LIN {X 0,Y 358.21,Z 356.559,A -85,B 0,C 180,E1 -13447.914,E2 -13447.914} C_VEL
LIN {X 0,Y 359.231,Z 351.066,A -85,B 0,C 180,E1 -13450.213,E2 -13450.213} C_VEL
LIN {X 0,Y 358.495,Z 346.197,A -85,B 0,C 180,E1 -13452.681,E2 -13452.681} C_VEL
LIN {X 0,Y 357.44,Z 341.043,A -85,B 0,C 180,E1 -13455.752,E2 -13455.752} C_VEL
LIN {X 0,Y 356.358,Z 336.09,A -85,B 0,C 180,E1 -13459.397,E2 -13459.397} C_VEL
LIN {X 0,Y 355.734,Z 333.05,A -85,B 0,C 180,E1 -13462.234,E2 -13462.234} C_VEL
LIN {X 0,Y 355.208,Z 330.772,A -85,B 0,C 180,E1 -13464.986,E2 -13464.986} C_VEL
LIN {X 0,Y 354.793,Z 328.931,A -85,B 0,C 180,E1 -13468.088,E2 -13468.088} C_VEL
LIN {X 0,Y 354.858,Z 329.119,A -85,B 0,C 180,E1 -13470.427,E2 -13470.427} C_VEL
LIN {X 0,Y 355.199,Z 330.372,A -85,B 0,C 180,E1 -13470.749,E2 -13470.749} C_VEL
LIN {X 0,Y 356.216,Z 332.283,A -85,B 0,C 180,E1 -13471.122,E2 -13471.122} C_VEL
LIN {X 0,Y 357.49,Z 333.609,A -85,B 0,C 180,E1 -13471.474,E2 -13471.474} C_VEL
LIN {X 0,Y 358.898,Z 336.455,A -85,B 0,C 180,E1 -13471.968,E2 -13471.968} C_VEL
LIN {X 0,Y 362.469,Z 342.56,A -85,B 0,C 180,E1 -13473.115,E2 -13473.115} C_VEL
LIN {X 0,Y 366.125,Z 350.503,A -85,B 0,C 180,E1 -13474.449,E2 -13474.449} C_VEL
LIN {X 0,Y 369.455,Z 359.944,A -85,B 0,C 180,E1 -13475.937,E2 -13475.937} C_VEL
LIN {X 0,Y 370.427,Z 363.82,A -85,B 0,C 180,E1 -13476.52,E2 -13476.52} C_VEL
LIN {X 0,Y 368.443,Z 376.173,A -85,B 0,C 180,E1 -13477.869,E2 -13477.869} C_VEL
LIN {X 0,Y 366.706,Z 386.37,A -85,B 0,C 180,E1 -13479.234,E2 -13479.234} C_VEL
LIN {X 0,Y 364.738,Z 396.604,A -85,B 0,C 180,E1 -13480.879,E2 -13480.879} C_VEL
LIN {X 0,Y 362.547,Z 406.465,A -85,B 0,C 180,E1 -13482.805,E2 -13482.805} C_VEL
LIN {X 0,Y 360.903,Z 414.416,A -85,B 0,C 180,E1 -13484.759,E2 -13484.759} C_VEL
LIN {X 0,Y 359.55,Z 419.998,A -85,B 0,C 180,E1 -13486.435,E2 -13486.435} C_VEL
LIN {X 0,Y 358.205,Z 425.911,A -85,B 0,C 180,E1 -13488.685,E2 -13488.685} C_VEL
LIN {X 0,Y 356.995,Z 430.235,A -85,B 0,C 180,E1 -13490.939,E2 -13490.939} C_VEL
LIN {X 0,Y 356.046,Z 433.125,A -85,B 0,C 180,E1 -13493.199,E2 -13493.199} C_VEL
LIN {X 0,Y 355.518,Z 434.622,A -85,B 0,C 180,E1 -13495.465,E2 -13495.465} C_VEL
LIN {X 0,Y 355.148,Z 434.801,A -85,B 0,C 180,E1 -13497.732,E2 -13497.732} C_VEL
LIN {X 0,Y 354.952,Z 433.645,A -85,B 0,C 180,E1 -13500,E2 -13500} C_VEL
LIN {X 0,Y 354.878,Z 431.132,A -85,B 0,C 180,E1 -13502.27,E2 -13502.27} C_VEL
LIN {X 0,Y 354.897,Z 427.195,A -85,B 0,C 180,E1 -13504.544,E2 -13504.544} C_VEL
LIN {X 0,Y 355.363,Z 423.255,A -85,B 0,C 180,E1 -13506.245,E2 -13506.245} C_VEL
LIN {X 0,Y 355.737,Z 418.361,A -85,B 0,C 180,E1 -13507.949,E2 -13507.949} C_VEL
LIN {X 0,Y 356.3,Z 411.398,A -85,B 0,C 180,E1 -13509.939,E2 -13509.939} C_VEL
LIN {X 0,Y 357.101,Z 402.834,A -85,B 0,C 180,E1 -13511.926,E2 -13511.926} C_VEL
LIN {X 0,Y 357.899,Z 393.943,A -85,B 0,C 180,E1 -13513.63,E2 -13513.63} C_VEL
LIN {X 0,Y 358.893,Z 383.272,A -85,B 0,C 180,E1 -13515.329,E2 -13515.329} C_VEL
LIN {X 0,Y 359.931,Z 372.22,A -85,B 0,C 180,E1 -13516.794,E2 -13516.794} C_VEL
LIN {X 0,Y 360.928,Z 359.901,A -85,B 0,C 180,E1 -13518.153,E2 -13518.153} C_VEL
LIN {X 0,Y 361.541,Z 352.454,A -85,B 0,C 180,E1 -13518.855,E2 -13518.855} C_VEL
LIN {X 0,Y 358.245,Z 340.353,A -85,B 0,C 180,E1 -13520.025,E2 -13520.025} C_VEL
LIN {X 0,Y 354.959,Z 329.484,A -85,B 0,C 180,E1 -13520.98,E2 -13520.98} C_VEL
LIN {X 0,Y 354.871,Z 328.937,A -85,B 0,C 180,E1 -13521.207,E2 -13521.207} C_VEL
LIN {X 0,Y 354.867,Z 328.909,A -85,B 0,C 180,E1 -13524.576,E2 -13524.576} C_VEL
LIN {X 0,Y 354.889,Z 328.902,A -85,B 0,C 180,E1 -13527.096,E2 -13527.096} C_VEL
LIN {X 0,Y 354.859,Z 328.904,A -85,B 0,C 180,E1 -13529.679,E2 -13529.679} C_VEL
LIN {X 0,Y 354.811,Z 328.91,A -85,B 0,C 180,E1 -13533.702,E2 -13533.702} C_VEL
LIN {X 0,Y 354.803,Z 328.916,A -85,B 0,C 180,E1 -13536.459,E2 -13536.459} C_VEL
LIN {X 0,Y 354.829,Z 328.907,A -85,B 0,C 180,E1 -13539.424,E2 -13539.424} C_VEL
LIN {X 0,Y 354.793,Z 328.914,A -85,B 0,C 180,E1 -13542.867,E2 -13542.867} C_VEL
LIN {X 0,Y 354.782,Z 328.916,A -85,B 0,C 180,E1 -13546.105,E2 -13546.105} C_VEL
LIN {X 0,Y 354.83,Z 328.908,A -85,B 0,C 180,E1 -13549.184,E2 -13549.184} C_VEL
LIN {X 0,Y 354.818,Z 328.914,A -85,B 0,C 180,E1 -13552.401,E2 -13552.401} C_VEL
LIN {X 0,Y 354.818,Z 328.91,A -85,B 0,C 180,E1 -13554.941,E2 -13554.941} C_VEL
LIN {X 0,Y 354.799,Z 328.916,A -85,B 0,C 180,E1 -13558.405,E2 -13558.405} C_VEL
LIN {X 0,Y 354.852,Z 328.906,A -85,B 0,C 180,E1 -13561.618,E2 -13561.618} C_VEL
LIN {X 0,Y 354.904,Z 328.904,A -85,B 0,C 180,E1 -13564.172,E2 -13564.172} C_VEL
LIN {X 0,Y 354.821,Z 328.913,A -85,B 0,C 180,E1 -13567.892,E2 -13567.892} C_VEL
LIN {X 0,Y 354.929,Z 328.9,A -85,B 0,C 180,E1 -13571.891,E2 -13571.891} C_VEL
LIN {X 0,Y 354.949,Z 328.899,A -85,B 0,C 180,E1 -13575.98,E2 -13575.98} C_VEL
LIN {X 0,Y 354.983,Z 328.893,A -85,B 0,C 180,E1 -13579.735,E2 -13579.735} C_VEL
LIN {X 0,Y 355.119,Z 328.876,A -85,B 0,C 180,E1 -13582.036,E2 -13582.036} C_VEL
LIN {X 0,Y 355.096,Z 328.876,A -85,B 0,C 180,E1 -13584.32,E2 -13584.32} C_VEL
LIN {X 0,Y 355.249,Z 328.861,A -85,B 0,C 180,E1 -13587.731,E2 -13587.731} C_VEL
LIN {X 0,Y 355.401,Z 328.84,A -85,B 0,C 180,E1 -13589.999,E2 -13589.999} C_VEL
LIN {X 0,Y 355.248,Z 328.856,A -85,B 0,C 180,E1 -13592.267,E2 -13592.267} C_VEL
LIN {X 0,Y 355.143,Z 328.869,A -85,B 0,C 180,E1 -13596.818,E2 -13596.818} C_VEL
LIN {X 0,Y 355.019,Z 328.885,A -85,B 0,C 180,E1 -13599.111,E2 -13599.111} C_VEL
LIN {X 0,Y 354.924,Z 328.896,A -85,B 0,C 180,E1 -13602.58,E2 -13602.58} C_VEL
LIN {X 0,Y 354.892,Z 328.901,A -85,B 0,C 180,E1 -13606.095,E2 -13606.095} C_VEL
LIN {X 0,Y 354.903,Z 328.898,A -85,B 0,C 180,E1 -13608.471,E2 -13608.471} C_VEL
LIN {X 0,Y 354.837,Z 328.907,A -85,B 0,C 180,E1 -13612.105,E2 -13612.105} C_VEL
LIN {X 0,Y 354.9,Z 328.9,A -85,B 0,C 180,E1 -13615.826,E2 -13615.826} C_VEL
LIN {X 0,Y 354.817,Z 328.911,A -85,B 0,C 180,E1 -13619.68,E2 -13619.68} C_VEL
LIN {X 0,Y 354.805,Z 328.912,A -85,B 0,C 180,E1 -13623.701,E2 -13623.701} C_VEL
LIN {X 0,Y 354.796,Z 328.912,A -85,B 0,C 180,E1 -13626.458,E2 -13626.458} C_VEL
LIN {X 0,Y 354.822,Z 328.912,A -85,B 0,C 180,E1 -13629.422,E2 -13629.422} C_VEL
LIN {X 0,Y 354.786,Z 328.917,A -85,B 0,C 180,E1 -13632.866,E2 -13632.866} C_VEL
LIN {X 0,Y 354.773,Z 328.914,A -85,B 0,C 180,E1 -13636.104,E2 -13636.104} C_VEL
LIN {X 0,Y 354.774,Z 328.916,A -85,B 0,C 180,E1 -13639.533,E2 -13639.533} C_VEL
LIN {X 0,Y 354.116,Z 329,A -85,B 0,C 180,E1 -13640.481,E2 -13640.481} C_VEL
LIN {X 0,Y 351.3,Z 329.347,A -85,B 0,C 180,E1 -13642.024,E2 -13642.024} C_VEL
LIN {X 0,Y 348.899,Z 329.649,A -85,B 0,C 180,E1 -13643.272,E2 -13643.272} C_VEL
LIN {X 0,Y 347.846,Z 329.778,A -85,B 0,C 180,E1 -13644.237,E2 -13644.237} C_VEL
LIN {X 0,Y 347.748,Z 329.787,A -85,B 0,C 180,E1 -13644.564,E2 -13644.564} C_VEL
LIN {X 0,Y 347.759,Z 329.789,A -85,B 0,C 180,E1 -13648.301,E2 -13648.301} C_VEL
LIN {X 0,Y 347.801,Z 329.787,A -85,B 0,C 180,E1 -13650.989,E2 -13650.989} C_VEL
LIN {X 0,Y 347.826,Z 329.78,A -85,B 0,C 180,E1 -13653.607,E2 -13653.607} C_VEL
LIN {X 0,Y 347.783,Z 329.786,A -85,B 0,C 180,E1 -13656.161,E2 -13656.161} C_VEL
LIN {X 0,Y 347.806,Z 329.783,A -85,B 0,C 180,E1 -13659.909,E2 -13659.909} C_VEL
LIN {X 0,Y 347.859,Z 329.779,A -85,B 0,C 180,E1 -13662.358,E2 -13662.358} C_VEL
LIN {X 0,Y 347.89,Z 329.773,A -85,B 0,C 180,E1 -13665.97,E2 -13665.97} C_VEL
LIN {X 0,Y 347.921,Z 329.768,A -85,B 0,C 180,E1 -13669.525,E2 -13669.525} C_VEL
LIN {X 0,Y 348.1,Z 329.747,A -85,B 0,C 180,E1 -13673.042,E2 -13673.042} C_VEL
LIN {X 0,Y 348.201,Z 329.734,A -85,B 0,C 180,E1 -13677.686,E2 -13677.686} C_VEL
LIN {X 0,Y 348.338,Z 329.718,A -85,B 0,C 180,E1 -13680,E2 -13680} C_VEL
LIN {X 0,Y 348.201,Z 329.739,A -85,B 0,C 180,E1 -13682.313,E2 -13682.313} C_VEL
LIN {X 0,Y 348.098,Z 329.747,A -85,B 0,C 180,E1 -13686.958,E2 -13686.958} C_VEL
LIN {X 0,Y 347.961,Z 329.763,A -85,B 0,C 180,E1 -13689.298,E2 -13689.298} C_VEL
LIN {X 0,Y 347.886,Z 329.773,A -85,B 0,C 180,E1 -13692.839,E2 -13692.839} C_VEL
LIN {X 0,Y 347.833,Z 329.782,A -85,B 0,C 180,E1 -13696.431,E2 -13696.431} C_VEL
LIN {X 0,Y 347.848,Z 329.777,A -85,B 0,C 180,E1 -13698.86,E2 -13698.86} C_VEL
LIN {X 0,Y 347.766,Z 329.789,A -85,B 0,C 180,E1 -13702.58,E2 -13702.58} C_VEL
LIN {X 0,Y 347.804,Z 329.783,A -85,B 0,C 180,E1 -13705.109,E2 -13705.109} C_VEL
LIN {X 0,Y 347.805,Z 329.786,A -85,B 0,C 180,E1 -13707.694,E2 -13707.694} C_VEL
LIN {X 0,Y 347.763,Z 329.79,A -85,B 0,C 180,E1 -13710.346,E2 -13710.346} C_VEL
LIN {X 0,Y 347.741,Z 329.795,A -85,B 0,C 180,E1 -13714.044,E2 -13714.044} C_VEL
LIN {X 0,Y 347.76,Z 329.793,A -85,B 0,C 180,E1 -13717.321,E2 -13717.321} C_VEL
LIN {X 0,Y 347.86,Z 330.034,A -85,B 0,C 180,E1 -13719.537,E2 -13719.537} C_VEL
LIN {X 0,Y 349.468,Z 338.436,A -85,B 0,C 180,E1 -13723.138,E2 -13723.138} C_VEL
LIN {X 0,Y 351.233,Z 347.023,A -85,B 0,C 180,E1 -13726.645,E2 -13726.645} C_VEL
LIN {X 0,Y 352.492,Z 353.68,A -85,B 0,C 180,E1 -13729.257,E2 -13729.257} C_VEL
LIN {X 0,Y 352.257,Z 357.86,A -85,B 0,C 180,E1 -13730.782,E2 -13730.782} C_VEL
LIN {X 0,Y 350.874,Z 368.306,A -85,B 0,C 180,E1 -13734.49,E2 -13734.49} C_VEL
LIN {X 0,Y 349.619,Z 379.808,A -85,B 0,C 180,E1 -13738.491,E2 -13738.491} C_VEL
LIN {X 0,Y 348.526,Z 391.621,A -85,B 0,C 180,E1 -13742.53,E2 -13742.53} C_VEL
LIN {X 0,Y 347.843,Z 402.269,A -85,B 0,C 180,E1 -13746.072,E2 -13746.072} C_VEL
LIN {X 0,Y 348.261,Z 406.952,A -85,B 0,C 180,E1 -13746.317,E2 -13746.317} C_VEL
LIN {X 0,Y 350.008,Z 423.225,A -85,B 0,C 180,E1 -13747.11,E2 -13747.11} C_VEL
LIN {X 0,Y 351.474,Z 437.917,A -85,B 0,C 180,E1 -13748.059,E2 -13748.059} C_VEL
LIN {X 0,Y 352.452,Z 450.642,A -85,B 0,C 180,E1 -13749.077,E2 -13749.077} C_VEL
LIN {X 0,Y 352.517,Z 455.971,A -85,B 0,C 180,E1 -13749.557,E2 -13749.557} C_VEL
LIN {X 0,Y 351.156,Z 468.911,A -85,B 0,C 180,E1 -13750.87,E2 -13750.87} C_VEL
LIN {X 0,Y 349.938,Z 480.529,A -85,B 0,C 180,E1 -13752.317,E2 -13752.317} C_VEL
LIN {X 0,Y 348.836,Z 491.162,A -85,B 0,C 180,E1 -13753.919,E2 -13753.919} C_VEL
LIN {X 0,Y 347.921,Z 500.982,A -85,B 0,C 180,E1 -13755.705,E2 -13755.705} C_VEL
LIN {X 0,Y 347.322,Z 510.138,A -85,B 0,C 180,E1 -13757.734,E2 -13757.734} C_VEL
LIN {X 0,Y 347.071,Z 516.625,A -85,B 0,C 180,E1 -13759.501,E2 -13759.501} C_VEL
LIN {X 0,Y 347.029,Z 521.956,A -85,B 0,C 180,E1 -13761.265,E2 -13761.265} C_VEL
LIN {X 0,Y 347.145,Z 526.251,A -85,B 0,C 180,E1 -13763.024,E2 -13763.024} C_VEL
LIN {X 0,Y 347.243,Z 528.547,A -85,B 0,C 180,E1 -13764.193,E2 -13764.193} C_VEL
LIN {X 0,Y 347.327,Z 530.421,A -85,B 0,C 180,E1 -13765.359,E2 -13765.359} C_VEL
LIN {X 0,Y 347.494,Z 532.968,A -85,B 0,C 180,E1 -13767.683,E2 -13767.683} C_VEL
LIN {X 0,Y 347.652,Z 533.671,A -85,B 0,C 180,E1 -13768.843,E2 -13768.843} C_VEL
LIN {X 0,Y 347.813,Z 533.994,A -85,B 0,C 180,E1 -13770.001,E2 -13770.001} C_VEL
LIN {X 0,Y 347.636,Z 533.883,A -85,B 0,C 180,E1 -13771.159,E2 -13771.159} C_VEL
LIN {X 0,Y 347.32,Z 532.528,A -85,B 0,C 180,E1 -13773.481,E2 -13773.481} C_VEL
LIN {X 0,Y 347.26,Z 531.296,A -85,B 0,C 180,E1 -13774.644,E2 -13774.644} C_VEL
LIN {X 0,Y 346.944,Z 527.65,A -85,B 0,C 180,E1 -13776.982,E2 -13776.982} C_VEL
LIN {X 0,Y 346.835,Z 522.461,A -85,B 0,C 180,E1 -13779.33,E2 -13779.33} C_VEL
LIN {X 0,Y 347.057,Z 515.657,A -85,B 0,C 180,E1 -13781.684,E2 -13781.684} C_VEL
LIN {X 0,Y 347.553,Z 508.19,A -85,B 0,C 180,E1 -13783.764,E2 -13783.764} C_VEL
LIN {X 0,Y 348.651,Z 499.382,A -85,B 0,C 180,E1 -13785.792,E2 -13785.792} C_VEL
LIN {X 0,Y 350.156,Z 488.785,A -85,B 0,C 180,E1 -13787.824,E2 -13787.824} C_VEL
LIN {X 0,Y 351.863,Z 478.059,A -85,B 0,C 180,E1 -13789.547,E2 -13789.547} C_VEL
LIN {X 0,Y 354.112,Z 465.669,A -85,B 0,C 180,E1 -13791.206,E2 -13791.206} C_VEL
LIN {X 0,Y 355.448,Z 457.007,A -85,B 0,C 180,E1 -13792.22,E2 -13792.22} C_VEL
LIN {X 0,Y 356.489,Z 442.001,A -85,B 0,C 180,E1 -13793.839,E2 -13793.839} C_VEL
LIN {X 0,Y 356.905,Z 429.081,A -85,B 0,C 180,E1 -13795.068,E2 -13795.068} C_VEL
LIN {X 0,Y 355.903,Z 414.715,A -85,B 0,C 180,E1 -13796.417,E2 -13796.417} C_VEL
LIN {X 0,Y 353.771,Z 400.728,A -85,B 0,C 180,E1 -13797.755,E2 -13797.755} C_VEL
LIN {X 0,Y 351.399,Z 390.456,A -85,B 0,C 180,E1 -13798.806,E2 -13798.806} C_VEL
LIN {X 0,Y 349.931,Z 384.822,A -85,B 0,C 180,E1 -13799.41,E2 -13799.41} C_VEL
LIN {X 0,Y 348.704,Z 379.658,A -85,B 0,C 180,E1 -13800.02,E2 -13800.02} C_VEL
LIN {X 0,Y 349.364,Z 371.354,A -85,B 0,C 180,E1 -13802.899,E2 -13802.899} C_VEL
LIN {X 0,Y 351.102,Z 359.077,A -85,B 0,C 180,E1 -13807.628,E2 -13807.628} C_VEL
LIN {X 0,Y 352.334,Z 353.05,A -85,B 0,C 180,E1 -13810.181,E2 -13810.181} C_VEL
LIN {X 0,Y 351.778,Z 348.823,A -85,B 0,C 180,E1 -13812.336,E2 -13812.336} C_VEL
LIN {X 0,Y 350.768,Z 343.559,A -85,B 0,C 180,E1 -13815.472,E2 -13815.472} C_VEL
LIN {X 0,Y 349.841,Z 339.385,A -85,B 0,C 180,E1 -13818.476,E2 -13818.476} C_VEL
LIN {X 0,Y 349.07,Z 335.73,A -85,B 0,C 180,E1 -13821.741,E2 -13821.741} C_VEL
LIN {X 0,Y 348.62,Z 333.528,A -85,B 0,C 180,E1 -13824.224,E2 -13824.224} C_VEL
LIN {X 0,Y 348.025,Z 331.094,A -85,B 0,C 180,E1 -13828.012,E2 -13828.012} C_VEL
LIN {X 0,Y 347.987,Z 330.832,A -85,B 0,C 180,E1 -13829.087,E2 -13829.087} C_VEL
LIN {X 0,Y 348.425,Z 331.95,A -85,B 0,C 180,E1 -13829.414,E2 -13829.414} C_VEL
LIN {X 0,Y 351.075,Z 335.588,A -85,B 0,C 180,E1 -13830.34,E2 -13830.34} C_VEL
LIN {X 0,Y 353.971,Z 340.403,A -85,B 0,C 180,E1 -13831.377,E2 -13831.377} C_VEL
LIN {X 0,Y 358.973,Z 349.987,A -85,B 0,C 180,E1 -13833.238,E2 -13833.238} C_VEL
LIN {X 0,Y 362.937,Z 360.351,A -85,B 0,C 180,E1 -13835.026,E2 -13835.026} C_VEL
LIN {X 0,Y 364.372,Z 365.464,A -85,B 0,C 180,E1 -13835.863,E2 -13835.863} C_VEL
LIN {X 0,Y 364.163,Z 368.887,A -85,B 0,C 180,E1 -13836.268,E2 -13836.268} C_VEL
LIN {X 0,Y 361.965,Z 381.279,A -85,B 0,C 180,E1 -13837.752,E2 -13837.752} C_VEL
LIN {X 0,Y 359.8,Z 392.578,A -85,B 0,C 180,E1 -13839.415,E2 -13839.415} C_VEL
LIN {X 0,Y 357.866,Z 401.378,A -85,B 0,C 180,E1 -13840.974,E2 -13840.974} C_VEL
LIN {X 0,Y 355.829,Z 409.806,A -85,B 0,C 180,E1 -13842.767,E2 -13842.767} C_VEL
LIN {X 0,Y 354.332,Z 416.343,A -85,B 0,C 180,E1 -13844.469,E2 -13844.469} C_VEL
LIN {X 0,Y 352.897,Z 421.787,A -85,B 0,C 180,E1 -13846.174,E2 -13846.174} C_VEL
LIN {X 0,Y 351.735,Z 426.232,A -85,B 0,C 180,E1 -13847.89,E2 -13847.89} C_VEL
LIN {X 0,Y 350.743,Z 429.795,A -85,B 0,C 180,E1 -13849.611,E2 -13849.611} C_VEL
LIN {X 0,Y 349.634,Z 433.266,A -85,B 0,C 180,E1 -13851.912,E2 -13851.912} C_VEL
LIN {X 0,Y 348.796,Z 435.346,A -85,B 0,C 180,E1 -13854.218,E2 -13854.218} C_VEL
LIN {X 0,Y 348.325,Z 436.073,A -85,B 0,C 180,E1 -13856.53,E2 -13856.53} C_VEL
LIN {X 0,Y 347.999,Z 435.482,A -85,B 0,C 180,E1 -13858.843,E2 -13858.843} C_VEL
LIN {X 0,Y 347.927,Z 433.515,A -85,B 0,C 180,E1 -13861.158,E2 -13861.158} C_VEL
LIN {X 0,Y 347.718,Z 430.201,A -85,B 0,C 180,E1 -13863.477,E2 -13863.477} C_VEL
LIN {X 0,Y 348.193,Z 425.374,A -85,B 0,C 180,E1 -13865.793,E2 -13865.793} C_VEL
LIN {X 0,Y 348.729,Z 418.977,A -85,B 0,C 180,E1 -13868.11,E2 -13868.11} C_VEL
LIN {X 0,Y 349.309,Z 412.005,A -85,B 0,C 180,E1 -13870.111,E2 -13870.111} C_VEL
LIN {X 0,Y 350.169,Z 403.159,A -85,B 0,C 180,E1 -13872.166,E2 -13872.166} C_VEL
LIN {X 0,Y 351,Z 394.131,A -85,B 0,C 180,E1 -13873.903,E2 -13873.903} C_VEL
LIN {X 0,Y 352.043,Z 383.296,A -85,B 0,C 180,E1 -13875.635,E2 -13875.635} C_VEL
LIN {X 0,Y 353.134,Z 371.516,A -85,B 0,C 180,E1 -13877.197,E2 -13877.197} C_VEL
LIN {X 0,Y 354.154,Z 359.525,A -85,B 0,C 180,E1 -13878.513,E2 -13878.513} C_VEL
LIN {X 0,Y 354.618,Z 353.609,A -85,B 0,C 180,E1 -13879.075,E2 -13879.075} C_VEL
LIN {X 0,Y 351.253,Z 341.576,A -85,B 0,C 180,E1 -13880.275,E2 -13880.275} C_VEL
LIN {X 0,Y 347.917,Z 330.342,A -85,B 0,C 180,E1 -13881.283,E2 -13881.283} C_VEL
LIN {X 0,Y 347.811,Z 329.819,A -85,B 0,C 180,E1 -13881.501,E2 -13881.501} C_VEL
LIN {X 0,Y 347.818,Z 329.783,A -85,B 0,C 180,E1 -13885.108,E2 -13885.108} C_VEL
LIN {X 0,Y 347.816,Z 329.781,A -85,B 0,C 180,E1 -13887.694,E2 -13887.694} C_VEL
LIN {X 0,Y 347.769,Z 329.79,A -85,B 0,C 180,E1 -13890.346,E2 -13890.346} C_VEL
LIN {X 0,Y 347.75,Z 329.794,A -85,B 0,C 180,E1 -13894.464,E2 -13894.464} C_VEL
LIN {X 0,Y 347.778,Z 329.787,A -85,B 0,C 180,E1 -13897.988,E2 -13897.988} C_VEL
LIN {X 0,Y 347.756,Z 329.789,A -85,B 0,C 180,E1 -13901.83,E2 -13901.83} C_VEL
LIN {X 0,Y 347.714,Z 329.795,A -85,B 0,C 180,E1 -13905.026,E2 -13905.026} C_VEL
LIN {X 0,Y 347.773,Z 329.793,A -85,B 0,C 180,E1 -13908.394,E2 -13908.394} C_VEL
LIN {X 0,Y 347.783,Z 329.788,A -85,B 0,C 180,E1 -13912.01,E2 -13912.01} C_VEL
LIN {X 0,Y 347.75,Z 329.79,A -85,B 0,C 180,E1 -13915.536,E2 -13915.536} C_VEL
LIN {X 0,Y 347.751,Z 329.795,A -85,B 0,C 180,E1 -13918.3,E2 -13918.3} C_VEL
LIN {X 0,Y 347.784,Z 329.785,A -85,B 0,C 180,E1 -13920.987,E2 -13920.987} C_VEL
LIN {X 0,Y 347.836,Z 329.78,A -85,B 0,C 180,E1 -13923.607,E2 -13923.607} C_VEL
LIN {X 0,Y 347.791,Z 329.79,A -85,B 0,C 180,E1 -13926.161,E2 -13926.161} C_VEL
LIN {X 0,Y 347.818,Z 329.786,A -85,B 0,C 180,E1 -13929.909,E2 -13929.909} C_VEL
LIN {X 0,Y 347.872,Z 329.777,A -85,B 0,C 180,E1 -13932.359,E2 -13932.359} C_VEL
LIN {X 0,Y 347.903,Z 329.776,A -85,B 0,C 180,E1 -13935.97,E2 -13935.97} C_VEL
LIN {X 0,Y 347.934,Z 329.769,A -85,B 0,C 180,E1 -13939.525,E2 -13939.525} C_VEL
LIN {X 0,Y 348.079,Z 329.755,A -85,B 0,C 180,E1 -13941.874,E2 -13941.874} C_VEL
LIN {X 0,Y 348.072,Z 329.752,A -85,B 0,C 180,E1 -13944.205,E2 -13944.205} C_VEL
LIN {X 0,Y 348.211,Z 329.737,A -85,B 0,C 180,E1 -13947.686,E2 -13947.686} C_VEL
LIN {X 0,Y 348.349,Z 329.718,A -85,B 0,C 180,E1 -13949.999,E2 -13949.999} C_VEL
LIN {X 0,Y 348.211,Z 329.733,A -85,B 0,C 180,E1 -13952.312,E2 -13952.312} C_VEL
LIN {X 0,Y 348.111,Z 329.745,A -85,B 0,C 180,E1 -13956.956,E2 -13956.956} C_VEL
LIN {X 0,Y 347.971,Z 329.765,A -85,B 0,C 180,E1 -13959.297,E2 -13959.297} C_VEL
LIN {X 0,Y 347.893,Z 329.772,A -85,B 0,C 180,E1 -13962.838,E2 -13962.838} C_VEL
LIN {X 0,Y 347.841,Z 329.778,A -85,B 0,C 180,E1 -13966.43,E2 -13966.43} C_VEL
LIN {X 0,Y 347.853,Z 329.778,A -85,B 0,C 180,E1 -13968.859,E2 -13968.859} C_VEL
LIN {X 0,Y 347.777,Z 329.786,A -85,B 0,C 180,E1 -13972.578,E2 -13972.578} C_VEL
LIN {X 0,Y 347.813,Z 329.785,A -85,B 0,C 180,E1 -13975.107,E2 -13975.107} C_VEL
LIN {X 0,Y 347.808,Z 329.785,A -85,B 0,C 180,E1 -13977.693,E2 -13977.693} C_VEL
LIN {X 0,Y 347.748,Z 329.79,A -85,B 0,C 180,E1 -13980.346,E2 -13980.346} C_VEL
LIN {X 0,Y 347.747,Z 329.79,A -85,B 0,C 180,E1 -13984.042,E2 -13984.042} C_VEL
LIN {X 0,Y 347.76,Z 329.793,A -85,B 0,C 180,E1 -13987.319,E2 -13987.319} C_VEL
LIN {X 0,Y 347.73,Z 329.792,A -85,B 0,C 180,E1 -13990.296,E2 -13990.296} C_VEL
LIN {X 0,Y 347.723,Z 329.796,A -85,B 0,C 180,E1 -13993.406,E2 -13993.406} C_VEL
LIN {X 0,Y 347.724,Z 329.795,A -85,B 0,C 180,E1 -13996.685,E2 -13996.685} C_VEL
LIN {X 0,Y 347.743,Z 329.79,A -85,B 0,C 180,E1 -14000.172,E2 -14000.172} C_VEL
LIN {X 0,Y 347.758,Z 329.792,A -85,B 0,C 180,E1 -14002.678,E2 -14002.678} C_VEL
LIN {X 0,Y 347.748,Z 329.787,A -85,B 0,C 180,E1 -14004.564,E2 -14004.564} C_VEL
LIN {X 0,Y 347.041,Z 329.879,A -85,B 0,C 180,E1 -14005.531,E2 -14005.531} C_VEL
LIN {X 0,Y 344.165,Z 330.24,A -85,B 0,C 180,E1 -14007.104,E2 -14007.104} C_VEL
LIN {X 0,Y 341.778,Z 330.536,A -85,B 0,C 180,E1 -14008.377,E2 -14008.377} C_VEL
LIN {X 0,Y 340.793,Z 330.658,A -85,B 0,C 180,E1 -14009.362,E2 -14009.362} C_VEL
LIN {X 0,Y 340.733,Z 330.664,A -85,B 0,C 180,E1 -14009.696,E2 -14009.696} C_VEL
LIN {X 0,Y 340.799,Z 330.659,A -85,B 0,C 180,E1 -14013.019,E2 -14013.019} C_VEL
LIN {X 0,Y 340.723,Z 330.669,A -85,B 0,C 180,E1 -14016.926,E2 -14016.926} C_VEL
LIN {X 0,Y 340.784,Z 330.663,A -85,B 0,C 180,E1 -14020.733,E2 -14020.733} C_VEL
LIN {X 0,Y 340.779,Z 330.659,A -85,B 0,C 180,E1 -14023.218,E2 -14023.218} C_VEL
LIN {X 0,Y 340.837,Z 330.654,A -85,B 0,C 180,E1 -14026.89,E2 -14026.89} C_VEL
LIN {X 0,Y 340.921,Z 330.646,A -85,B 0,C 180,E1 -14030.507,E2 -14030.507} C_VEL
LIN {X 0,Y 341.07,Z 330.624,A -85,B 0,C 180,E1 -14032.898,E2 -14032.898} C_VEL
LIN {X 0,Y 341.163,Z 330.61,A -85,B 0,C 180,E1 -14037.638,E2 -14037.638} C_VEL
LIN {X 0,Y 341.289,Z 330.597,A -85,B 0,C 180,E1 -14040,E2 -14040} C_VEL
LIN {X 0,Y 341.163,Z 330.616,A -85,B 0,C 180,E1 -14042.361,E2 -14042.361} C_VEL
LIN {X 0,Y 341.067,Z 330.622,A -85,B 0,C 180,E1 -14047.102,E2 -14047.102} C_VEL
LIN {X 0,Y 340.867,Z 330.648,A -85,B 0,C 180,E1 -14050.694,E2 -14050.694} C_VEL
LIN {X 0,Y 340.855,Z 330.653,A -85,B 0,C 180,E1 -14054.325,E2 -14054.325} C_VEL
LIN {X 0,Y 340.83,Z 330.654,A -85,B 0,C 180,E1 -14058.467,E2 -14058.467} C_VEL
LIN {X 0,Y 340.746,Z 330.666,A -85,B 0,C 180,E1 -14061.857,E2 -14061.857} C_VEL
LIN {X 0,Y 340.765,Z 330.662,A -85,B 0,C 180,E1 -14065.665,E2 -14065.665} C_VEL
LIN {X 0,Y 340.735,Z 330.666,A -85,B 0,C 180,E1 -14068.32,E2 -14068.32} C_VEL
LIN {X 0,Y 340.709,Z 330.667,A -85,B 0,C 180,E1 -14071.043,E2 -14071.043} C_VEL
LIN {X 0,Y 340.712,Z 330.667,A -85,B 0,C 180,E1 -14075.279,E2 -14075.279} C_VEL
LIN {X 0,Y 340.757,Z 330.777,A -85,B 0,C 180,E1 -14079.103,E2 -14079.103} C_VEL
LIN {X 0,Y 342.317,Z 338.804,A -85,B 0,C 180,E1 -14082.649,E2 -14082.649} C_VEL
LIN {X 0,Y 344.21,Z 348.135,A -85,B 0,C 180,E1 -14086.548,E2 -14086.548} C_VEL
LIN {X 0,Y 345.37,Z 353.864,A -85,B 0,C 180,E1 -14088.844,E2 -14088.844} C_VEL
LIN {X 0,Y 345.438,Z 357.153,A -85,B 0,C 180,E1 -14090.098,E2 -14090.098} C_VEL
LIN {X 0,Y 344.144,Z 366.99,A -85,B 0,C 180,E1 -14093.686,E2 -14093.686} C_VEL
LIN {X 0,Y 342.762,Z 378.488,A -85,B 0,C 180,E1 -14097.786,E2 -14097.786} C_VEL
LIN {X 0,Y 341.62,Z 389.819,A -85,B 0,C 180,E1 -14101.761,E2 -14101.761} C_VEL
LIN {X 0,Y 340.85,Z 401.262,A -85,B 0,C 180,E1 -14105.687,E2 -14105.687} C_VEL
LIN {X 0,Y 340.886,Z 402.791,A -85,B 0,C 180,E1 -14105.832,E2 -14105.832} C_VEL
LIN {X 0,Y 342.64,Z 419.445,A -85,B 0,C 180,E1 -14106.626,E2 -14106.626} C_VEL
LIN {X 0,Y 344.141,Z 434.532,A -85,B 0,C 180,E1 -14107.584,E2 -14107.584} C_VEL
LIN {X 0,Y 345.253,Z 447.844,A -85,B 0,C 180,E1 -14108.64,E2 -14108.64} C_VEL
LIN {X 0,Y 345.548,Z 455.332,A -85,B 0,C 180,E1 -14109.322,E2 -14109.322} C_VEL
LIN {X 0,Y 344.227,Z 467.852,A -85,B 0,C 180,E1 -14110.625,E2 -14110.625} C_VEL
LIN {X 0,Y 342.971,Z 479.456,A -85,B 0,C 180,E1 -14112.1,E2 -14112.1} C_VEL
LIN {X 0,Y 341.742,Z 490.963,A -85,B 0,C 180,E1 -14113.882,E2 -14113.882} C_VEL
LIN {X 0,Y 340.814,Z 500.818,A -85,B 0,C 180,E1 -14115.742,E2 -14115.742} C_VEL
LIN {X 0,Y 340.263,Z 509.656,A -85,B 0,C 180,E1 -14117.779,E2 -14117.779} C_VEL
LIN {X 0,Y 339.993,Z 516.987,A -85,B 0,C 180,E1 -14119.882,E2 -14119.882} C_VEL
LIN {X 0,Y 340.022,Z 522.083,A -85,B 0,C 180,E1 -14121.682,E2 -14121.682} C_VEL
LIN {X 0,Y 340.17,Z 526.09,A -85,B 0,C 180,E1 -14123.476,E2 -14123.476} C_VEL
LIN {X 0,Y 340.298,Z 529.128,A -85,B 0,C 180,E1 -14125.263,E2 -14125.263} C_VEL
LIN {X 0,Y 340.496,Z 531.754,A -85,B 0,C 180,E1 -14127.635,E2 -14127.635} C_VEL
LIN {X 0,Y 340.653,Z 532.492,A -85,B 0,C 180,E1 -14128.819,E2 -14128.819} C_VEL
LIN {X 0,Y 340.802,Z 532.845,A -85,B 0,C 180,E1 -14130.001,E2 -14130.001} C_VEL
LIN {X 0,Y 340.633,Z 532.765,A -85,B 0,C 180,E1 -14131.183,E2 -14131.183} C_VEL
LIN {X 0,Y 340.275,Z 531.471,A -85,B 0,C 180,E1 -14133.553,E2 -14133.553} C_VEL
LIN {X 0,Y 340.187,Z 530.275,A -85,B 0,C 180,E1 -14134.741,E2 -14134.741} C_VEL
LIN {X 0,Y 339.878,Z 526.725,A -85,B 0,C 180,E1 -14137.128,E2 -14137.128} C_VEL
LIN {X 0,Y 339.746,Z 521.625,A -85,B 0,C 180,E1 -14139.527,E2 -14139.527} C_VEL
LIN {X 0,Y 340.002,Z 514.918,A -85,B 0,C 180,E1 -14141.93,E2 -14141.93} C_VEL
LIN {X 0,Y 340.734,Z 506.98,A -85,B 0,C 180,E1 -14144.205,E2 -14144.205} C_VEL
LIN {X 0,Y 341.915,Z 497.555,A -85,B 0,C 180,E1 -14146.418,E2 -14146.418} C_VEL
LIN {X 0,Y 343.644,Z 486.924,A -85,B 0,C 180,E1 -14148.482,E2 -14148.482} C_VEL
LIN {X 0,Y 345.731,Z 474.738,A -85,B 0,C 180,E1 -14150.443,E2 -14150.443} C_VEL
LIN {X 0,Y 348.441,Z 461.231,A -85,B 0,C 180,E1 -14152.222,E2 -14152.222} C_VEL
LIN {X 0,Y 349.877,Z 446.061,A -85,B 0,C 180,E1 -14154.003,E2 -14154.003} C_VEL
LIN {X 0,Y 350.724,Z 432.757,A -85,B 0,C 180,E1 -14155.364,E2 -14155.364} C_VEL
LIN {X 0,Y 350.267,Z 419.737,A -85,B 0,C 180,E1 -14156.674,E2 -14156.674} C_VEL
LIN {X 0,Y 348.912,Z 407.891,A -85,B 0,C 180,E1 -14157.876,E2 -14157.876} C_VEL
LIN {X 0,Y 346.501,Z 394.684,A -85,B 0,C 180,E1 -14159.29,E2 -14159.29} C_VEL
LIN {X 0,Y 344.818,Z 387.882,A -85,B 0,C 180,E1 -14160.084,E2 -14160.084} C_VEL
LIN {X 0,Y 343.493,Z 382.743,A -85,B 0,C 180,E1 -14160.7,E2 -14160.7} C_VEL
LIN {X 0,Y 342.149,Z 378.124,A -85,B 0,C 180,E1 -14161.308,E2 -14161.308} C_VEL
LIN {X 0,Y 342.042,Z 376.409,A -85,B 0,C 180,E1 -14161.599,E2 -14161.599} C_VEL
LIN {X 0,Y 343.236,Z 365.625,A -85,B 0,C 180,E1 -14165.702,E2 -14165.702} C_VEL
LIN {X 0,Y 345.023,Z 356.983,A -85,B 0,C 180,E1 -14169.282,E2 -14169.282} C_VEL
LIN {X 0,Y 345.457,Z 354.055,A -85,B 0,C 180,E1 -14170.619,E2 -14170.619} C_VEL
LIN {X 0,Y 344.838,Z 350,A -85,B 0,C 180,E1 -14172.803,E2 -14172.803} C_VEL
LIN {X 0,Y 343.823,Z 344.916,A -85,B 0,C 180,E1 -14175.974,E2 -14175.974} C_VEL
LIN {X 0,Y 342.848,Z 340.515,A -85,B 0,C 180,E1 -14179.33,E2 -14179.33} C_VEL
LIN {X 0,Y 342.26,Z 337.704,A -85,B 0,C 180,E1 -14181.974,E2 -14181.974} C_VEL
LIN {X 0,Y 341.658,Z 334.893,A -85,B 0,C 180,E1 -14185.368,E2 -14185.368} C_VEL
LIN {X 0,Y 341.374,Z 333.716,A -85,B 0,C 180,E1 -14187.575,E2 -14187.575} C_VEL
LIN {X 0,Y 341.884,Z 334.656,A -85,B 0,C 180,E1 -14187.991,E2 -14187.991} C_VEL
LIN {X 0,Y 344.527,Z 337.177,A -85,B 0,C 180,E1 -14188.956,E2 -14188.956} C_VEL
LIN {X 0,Y 349.322,Z 344.784,A -85,B 0,C 180,E1 -14190.849,E2 -14190.849} C_VEL
LIN {X 0,Y 354.04,Z 354.414,A -85,B 0,C 180,E1 -14192.834,E2 -14192.834} C_VEL
LIN {X 0,Y 357.637,Z 364.528,A -85,B 0,C 180,E1 -14194.684,E2 -14194.684} C_VEL
LIN {X 0,Y 358.704,Z 369.549,A -85,B 0,C 180,E1 -14195.522,E2 -14195.522} C_VEL
LIN {X 0,Y 356.262,Z 382.292,A -85,B 0,C 180,E1 -14197.07,E2 -14197.07} C_VEL
LIN {X 0,Y 353.948,Z 393.533,A -85,B 0,C 180,E1 -14198.754,E2 -14198.754} C_VEL
LIN {X 0,Y 351.691,Z 403.104,A -85,B 0,C 180,E1 -14200.485,E2 -14200.485} C_VEL
LIN {X 0,Y 349.376,Z 411.94,A -85,B 0,C 180,E1 -14202.438,E2 -14202.438} C_VEL
LIN {X 0,Y 347.766,Z 418.298,A -85,B 0,C 180,E1 -14204.168,E2 -14204.168} C_VEL
LIN {X 0,Y 346.265,Z 423.616,A -85,B 0,C 180,E1 -14205.904,E2 -14205.904} C_VEL
LIN {X 0,Y 344.677,Z 429.154,A -85,B 0,C 180,E1 -14208.235,E2 -14208.235} C_VEL
LIN {X 0,Y 343.29,Z 433.22,A -85,B 0,C 180,E1 -14210.574,E2 -14210.574} C_VEL
LIN {X 0,Y 342.242,Z 435.857,A -85,B 0,C 180,E1 -14212.923,E2 -14212.923} C_VEL
LIN {X 0,Y 341.589,Z 437.132,A -85,B 0,C 180,E1 -14215.28,E2 -14215.28} C_VEL
LIN {X 0,Y 341.14,Z 437.082,A -85,B 0,C 180,E1 -14217.639,E2 -14217.639} C_VEL
LIN {X 0,Y 340.914,Z 435.671,A -85,B 0,C 180,E1 -14220,E2 -14220} C_VEL
LIN {X 0,Y 340.826,Z 432.911,A -85,B 0,C 180,E1 -14222.364,E2 -14222.364} C_VEL
LIN {X 0,Y 340.786,Z 429.963,A -85,B 0,C 180,E1 -14224.14,E2 -14224.14} C_VEL
LIN {X 0,Y 341.188,Z 426.083,A -85,B 0,C 180,E1 -14225.912,E2 -14225.912} C_VEL
LIN {X 0,Y 341.722,Z 419.566,A -85,B 0,C 180,E1 -14228.278,E2 -14228.278} C_VEL
LIN {X 0,Y 342.326,Z 412.453,A -85,B 0,C 180,E1 -14230.319,E2 -14230.319} C_VEL
LIN {X 0,Y 343.24,Z 403.435,A -85,B 0,C 180,E1 -14232.415,E2 -14232.415} C_VEL
LIN {X 0,Y 344.081,Z 394.25,A -85,B 0,C 180,E1 -14234.188,E2 -14234.188} C_VEL
LIN {X 0,Y 345.196,Z 383.252,A -85,B 0,C 180,E1 -14235.954,E2 -14235.954} C_VEL
LIN {X 0,Y 346.342,Z 371.092,A -85,B 0,C 180,E1 -14237.57,E2 -14237.57} C_VEL
LIN {X 0,Y 347.423,Z 357.736,A -85,B 0,C 180,E1 -14239.014,E2 -14239.014} C_VEL
LIN {X 0,Y 347.476,Z 353.837,A -85,B 0,C 180,E1 -14239.4,E2 -14239.4} C_VEL
LIN {X 0,Y 343.721,Z 340.853,A -85,B 0,C 180,E1 -14240.699,E2 -14240.699} C_VEL
LIN {X 0,Y 340.865,Z 331.275,A -85,B 0,C 180,E1 -14241.574,E2 -14241.574} C_VEL
LIN {X 0,Y 340.759,Z 330.683,A -85,B 0,C 180,E1 -14241.857,E2 -14241.857} C_VEL
LIN {X 0,Y 340.778,Z 330.658,A -85,B 0,C 180,E1 -14245.664,E2 -14245.664} C_VEL
LIN {X 0,Y 340.746,Z 330.664,A -85,B 0,C 180,E1 -14248.32,E2 -14248.32} C_VEL
LIN {X 0,Y 340.709,Z 330.669,A -85,B 0,C 180,E1 -14251.044,E2 -14251.044} C_VEL
LIN {X 0,Y 340.723,Z 330.665,A -85,B 0,C 180,E1 -14255.279,E2 -14255.279} C_VEL
LIN {X 0,Y 340.715,Z 330.67,A -85,B 0,C 180,E1 -14258.386,E2 -14258.386} C_VEL
LIN {X 0,Y 340.704,Z 330.669,A -85,B 0,C 180,E1 -14262.045,E2 -14262.045} C_VEL
LIN {X 0,Y 340.673,Z 330.675,A -85,B 0,C 180,E1 -14266.224,E2 -14266.224} C_VEL
LIN {X 0,Y 340.71,Z 330.669,A -85,B 0,C 180,E1 -14268.693,E2 -14268.693} C_VEL
LIN {X 0,Y 340.743,Z 330.664,A -85,B 0,C 180,E1 -14271.773,E2 -14271.773} C_VEL
LIN {X 0,Y 340.729,Z 330.665,A -85,B 0,C 180,E1 -14275.595,E2 -14275.595} C_VEL
LIN {X 0,Y 340.704,Z 330.668,A -85,B 0,C 180,E1 -14278.955,E2 -14278.955} C_VEL
LIN {X 0,Y 340.809,Z 330.654,A -85,B 0,C 180,E1 -14283.019,E2 -14283.019} C_VEL
LIN {X 0,Y 340.76,Z 330.662,A -85,B 0,C 180,E1 -14285.638,E2 -14285.638} C_VEL
LIN {X 0,Y 340.743,Z 330.663,A -85,B 0,C 180,E1 -14289.473,E2 -14289.473} C_VEL
LIN {X 0,Y 340.864,Z 330.653,A -85,B 0,C 180,E1 -14291.984,E2 -14291.984} C_VEL
LIN {X 0,Y 340.875,Z 330.649,A -85,B 0,C 180,E1 -14295.704,E2 -14295.704} C_VEL
LIN {X 0,Y 340.876,Z 330.647,A -85,B 0,C 180,E1 -14299.305,E2 -14299.305} C_VEL
LIN {X 0,Y 341.08,Z 330.62,A -85,B 0,C 180,E1 -14302.897,E2 -14302.897} C_VEL
LIN {X 0,Y 341.173,Z 330.613,A -85,B 0,C 180,E1 -14307.638,E2 -14307.638} C_VEL
LIN {X 0,Y 341.3,Z 330.596,A -85,B 0,C 180,E1 -14309.999,E2 -14309.999} C_VEL
LIN {X 0,Y 341.173,Z 330.609,A -85,B 0,C 180,E1 -14312.36,E2 -14312.36} C_VEL
LIN {X 0,Y 341.08,Z 330.622,A -85,B 0,C 180,E1 -14317.101,E2 -14317.101} C_VEL
LIN {X 0,Y 340.874,Z 330.646,A -85,B 0,C 180,E1 -14320.692,E2 -14320.692} C_VEL
LIN {X 0,Y 340.865,Z 330.647,A -85,B 0,C 180,E1 -14324.324,E2 -14324.324} C_VEL
LIN {X 0,Y 340.839,Z 330.65,A -85,B 0,C 180,E1 -14328.465,E2 -14328.465} C_VEL
LIN {X 0,Y 340.755,Z 330.663,A -85,B 0,C 180,E1 -14331.855,E2 -14331.855} C_VEL
LIN {X 0,Y 340.773,Z 330.661,A -85,B 0,C 180,E1 -14335.663,E2 -14335.663} C_VEL
LIN {X 0,Y 340.728,Z 330.664,A -85,B 0,C 180,E1 -14338.319,E2 -14338.319} C_VEL
LIN {X 0,Y 340.697,Z 330.672,A -85,B 0,C 180,E1 -14341.043,E2 -14341.043} C_VEL
LIN {X 0,Y 340.716,Z 330.671,A -85,B 0,C 180,E1 -14345.277,E2 -14345.277} C_VEL
LIN {X 0,Y 340.708,Z 330.667,A -85,B 0,C 180,E1 -14348.385,E2 -14348.385} C_VEL
LIN {X 0,Y 340.696,Z 330.668,A -85,B 0,C 180,E1 -14352.044,E2 -14352.044} C_VEL
LIN {X 0,Y 340.68,Z 330.672,A -85,B 0,C 180,E1 -14355.46,E2 -14355.46} C_VEL
LIN {X 0,Y 340.683,Z 330.673,A -85,B 0,C 180,E1 -14358.689,E2 -14358.689} C_VEL
LIN {X 0,Y 340.729,Z 330.664,A -85,B 0,C 180,E1 -14361.772,E2 -14361.772} C_VEL
LIN {X 0,Y 340.718,Z 330.666,A -85,B 0,C 180,E1 -14365.594,E2 -14365.594} C_VEL
LIN {X 0,Y 340.733,Z 330.664,A -85,B 0,C 180,E1 -14369.696,E2 -14369.696} C_VEL
LIN {X 0,Y 340.112,Z 330.745,A -85,B 0,C 180,E1 -14370.682,E2 -14370.682} C_VEL
LIN {X 0,Y 337.254,Z 331.106,A -85,B 0,C 180,E1 -14372.286,E2 -14372.286} C_VEL
LIN {X 0,Y 334.816,Z 331.412,A -85,B 0,C 180,E1 -14373.585,E2 -14373.585} C_VEL
LIN {X 0,Y 333.786,Z 331.536,A -85,B 0,C 180,E1 -14374.591,E2 -14374.591} C_VEL
LIN {X 0,Y 333.714,Z 331.542,A -85,B 0,C 180,E1 -14374.932,E2 -14374.932} C_VEL
LIN {X 0,Y 333.679,Z 331.545,A -85,B 0,C 180,E1 -14379.019,E2 -14379.019} C_VEL
LIN {X 0,Y 333.787,Z 331.529,A -85,B 0,C 180,E1 -14381.589,E2 -14381.589} C_VEL
LIN {X 0,Y 333.801,Z 331.527,A -85,B 0,C 180,E1 -14385.576,E2 -14385.576} C_VEL
LIN {X 0,Y 333.826,Z 331.525,A -85,B 0,C 180,E1 -14389.077,E2 -14389.077} C_VEL
LIN {X 0,Y 334.019,Z 331.503,A -85,B 0,C 180,E1 -14392.747,E2 -14392.747} C_VEL
LIN {X 0,Y 333.806,Z 331.527,A -85,B 0,C 180,E1 -14395.169,E2 -14395.169} C_VEL
LIN {X 0,Y 334.1,Z 331.49,A -85,B 0,C 180,E1 -14397.588,E2 -14397.588} C_VEL
LIN {X 0,Y 334.239,Z 331.475,A -85,B 0,C 180,E1 -14400,E2 -14400} C_VEL
LIN {X 0,Y 334.1,Z 331.495,A -85,B 0,C 180,E1 -14402.411,E2 -14402.411} C_VEL
LIN {X 0,Y 334.017,Z 331.5,A -85,B 0,C 180,E1 -14407.252,E2 -14407.252} C_VEL
LIN {X 0,Y 333.829,Z 331.524,A -85,B 0,C 180,E1 -14410.922,E2 -14410.922} C_VEL
LIN {X 0,Y 333.8,Z 331.529,A -85,B 0,C 180,E1 -14414.634,E2 -14414.634} C_VEL
LIN {X 0,Y 333.789,Z 331.53,A -85,B 0,C 180,E1 -14418.656,E2 -14418.656} C_VEL
LIN {X 0,Y 333.684,Z 331.545,A -85,B 0,C 180,E1 -14422.278,E2 -14422.278} C_VEL
LIN {X 0,Y 333.728,Z 331.539,A -85,B 0,C 180,E1 -14426.247,E2 -14426.247} C_VEL
LIN {X 0,Y 333.704,Z 331.539,A -85,B 0,C 180,E1 -14428.972,E2 -14428.972} C_VEL
LIN {X 0,Y 333.644,Z 331.547,A -85,B 0,C 180,E1 -14432.59,E2 -14432.59} C_VEL
LIN {X 0,Y 333.671,Z 331.548,A -85,B 0,C 180,E1 -14436.139,E2 -14436.139} C_VEL
LIN {X 0,Y 333.726,Z 331.747,A -85,B 0,C 180,E1 -14438.816,E2 -14438.816} C_VEL
LIN {X 0,Y 335.177,Z 339.137,A -85,B 0,C 180,E1 -14442.142,E2 -14442.142} C_VEL
LIN {X 0,Y 337.236,Z 349.466,A -85,B 0,C 180,E1 -14446.552,E2 -14446.552} C_VEL
LIN {X 0,Y 338.465,Z 355.992,A -85,B 0,C 180,E1 -14449.207,E2 -14449.207} C_VEL
LIN {X 0,Y 338.122,Z 360.197,A -85,B 0,C 180,E1 -14450.808,E2 -14450.808} C_VEL
LIN {X 0,Y 336.722,Z 370.133,A -85,B 0,C 180,E1 -14454.488,E2 -14454.488} C_VEL
LIN {X 0,Y 335.481,Z 380.917,A -85,B 0,C 180,E1 -14458.419,E2 -14458.419} C_VEL
LIN {X 0,Y 334.353,Z 392.185,A -85,B 0,C 180,E1 -14462.457,E2 -14462.457} C_VEL
LIN {X 0,Y 333.802,Z 400.657,A -85,B 0,C 180,E1 -14465.389,E2 -14465.389} C_VEL
LIN {X 0,Y 334.54,Z 408.487,A -85,B 0,C 180,E1 -14465.777,E2 -14465.777} C_VEL
LIN {X 0,Y 336.023,Z 423.514,A -85,B 0,C 180,E1 -14466.586,E2 -14466.586} C_VEL
LIN {X 0,Y 337.409,Z 437.802,A -85,B 0,C 180,E1 -14467.594,E2 -14467.594} C_VEL
LIN {X 0,Y 338.378,Z 450.872,A -85,B 0,C 180,E1 -14468.724,E2 -14468.724} C_VEL
LIN {X 0,Y 338.355,Z 457.016,A -85,B 0,C 180,E1 -14469.324,E2 -14469.324} C_VEL
LIN {X 0,Y 337.007,Z 469.168,A -85,B 0,C 180,E1 -14470.668,E2 -14470.668} C_VEL
LIN {X 0,Y 335.77,Z 480.396,A -85,B 0,C 180,E1 -14472.176,E2 -14472.176} C_VEL
LIN {X 0,Y 334.665,Z 490.713,A -85,B 0,C 180,E1 -14473.845,E2 -14473.845} C_VEL
LIN {X 0,Y 333.718,Z 500.78,A -85,B 0,C 180,E1 -14475.82,E2 -14475.82} C_VEL
LIN {X 0,Y 333.198,Z 509.11,A -85,B 0,C 180,E1 -14477.825,E2 -14477.825} C_VEL
LIN {X 0,Y 332.957,Z 515.427,A -85,B 0,C 180,E1 -14479.665,E2 -14479.665} C_VEL
LIN {X 0,Y 332.983,Z 520.582,A -85,B 0,C 180,E1 -14481.505,E2 -14481.505} C_VEL
LIN {X 0,Y 333.154,Z 524.687,A -85,B 0,C 180,E1 -14483.338,E2 -14483.338} C_VEL
LIN {X 0,Y 333.269,Z 527.812,A -85,B 0,C 180,E1 -14485.162,E2 -14485.162} C_VEL
LIN {X 0,Y 333.494,Z 530.524,A -85,B 0,C 180,E1 -14487.586,E2 -14487.586} C_VEL
LIN {X 0,Y 333.652,Z 531.299,A -85,B 0,C 180,E1 -14488.794,E2 -14488.794} C_VEL
LIN {X 0,Y 333.793,Z 531.685,A -85,B 0,C 180,E1 -14490.001,E2 -14490.001} C_VEL
LIN {X 0,Y 333.626,Z 531.639,A -85,B 0,C 180,E1 -14491.208,E2 -14491.208} C_VEL
LIN {X 0,Y 333.228,Z 530.411,A -85,B 0,C 180,E1 -14493.629,E2 -14493.629} C_VEL
LIN {X 0,Y 333.116,Z 529.249,A -85,B 0,C 180,E1 -14494.842,E2 -14494.842} C_VEL
LIN {X 0,Y 332.791,Z 525.774,A -85,B 0,C 180,E1 -14497.281,E2 -14497.281} C_VEL
LIN {X 0,Y 332.674,Z 520.794,A -85,B 0,C 180,E1 -14499.731,E2 -14499.731} C_VEL
LIN {X 0,Y 332.96,Z 514.217,A -85,B 0,C 180,E1 -14502.186,E2 -14502.186} C_VEL
LIN {X 0,Y 333.816,Z 505.941,A -85,B 0,C 180,E1 -14504.635,E2 -14504.635} C_VEL
LIN {X 0,Y 335.246,Z 495.8,A -85,B 0,C 180,E1 -14507.068,E2 -14507.068} C_VEL
LIN {X 0,Y 337.183,Z 485.155,A -85,B 0,C 180,E1 -14509.166,E2 -14509.166} C_VEL
LIN {X 0,Y 339.33,Z 473.878,A -85,B 0,C 180,E1 -14511.021,E2 -14511.021} C_VEL
LIN {X 0,Y 342.089,Z 460.694,A -85,B 0,C 180,E1 -14512.817,E2 -14512.817} C_VEL
LIN {X 0,Y 343.626,Z 445.931,A -85,B 0,C 180,E1 -14514.629,E2 -14514.629} C_VEL
LIN {X 0,Y 344.557,Z 434.009,A -85,B 0,C 180,E1 -14515.915,E2 -14515.915} C_VEL
LIN {X 0,Y 344.295,Z 420.679,A -85,B 0,C 180,E1 -14517.34,E2 -14517.34} C_VEL
LIN {X 0,Y 342.703,Z 405.92,A -85,B 0,C 180,E1 -14518.966,E2 -14518.966} C_VEL
LIN {X 0,Y 340.167,Z 392.377,A -85,B 0,C 180,E1 -14520.577,E2 -14520.577} C_VEL
LIN {X 0,Y 338.684,Z 386.389,A -85,B 0,C 180,E1 -14521.369,E2 -14521.369} C_VEL
LIN {X 0,Y 337.041,Z 380.07,A -85,B 0,C 180,E1 -14522.231,E2 -14522.231} C_VEL
LIN {X 0,Y 335.621,Z 375.095,A -85,B 0,C 180,E1 -14522.988,E2 -14522.988} C_VEL
LIN {X 0,Y 335.512,Z 373.23,A -85,B 0,C 180,E1 -14523.358,E2 -14523.358} C_VEL
LIN {X 0,Y 337.387,Z 361.712,A -85,B 0,C 180,E1 -14528.052,E2 -14528.052} C_VEL
LIN {X 0,Y 338.487,Z 357.148,A -85,B 0,C 180,E1 -14530.066,E2 -14530.066} C_VEL
LIN {X 0,Y 338.382,Z 354.043,A -85,B 0,C 180,E1 -14531.654,E2 -14531.654} C_VEL
LIN {X 0,Y 337.375,Z 348.604,A -85,B 0,C 180,E1 -14534.906,E2 -14534.906} C_VEL
LIN {X 0,Y 336.41,Z 344.242,A -85,B 0,C 180,E1 -14538.047,E2 -14538.047} C_VEL
LIN {X 0,Y 335.705,Z 340.765,A -85,B 0,C 180,E1 -14541.094,E2 -14541.094} C_VEL
LIN {X 0,Y 334.998,Z 337.438,A -85,B 0,C 180,E1 -14544.905,E2 -14544.905} C_VEL
LIN {X 0,Y 334.894,Z 336.955,A -85,B 0,C 180,E1 -14545.85,E2 -14545.85} C_VEL
LIN {X 0,Y 335.232,Z 337.669,A -85,B 0,C 180,E1 -14546.252,E2 -14546.252} C_VEL
LIN {X 0,Y 338.485,Z 340.565,A -85,B 0,C 180,E1 -14547.658,E2 -14547.658} C_VEL
LIN {X 0,Y 341.232,Z 343.547,A -85,B 0,C 180,E1 -14548.781,E2 -14548.781} C_VEL
LIN {X 0,Y 345.307,Z 350.58,A -85,B 0,C 180,E1 -14550.6,E2 -14550.6} C_VEL
LIN {X 0,Y 349.098,Z 358.843,A -85,B 0,C 180,E1 -14552.417,E2 -14552.417} C_VEL
LIN {X 0,Y 352.216,Z 368.313,A -85,B 0,C 180,E1 -14554.266,E2 -14554.266} C_VEL
LIN {X 0,Y 352.986,Z 371.739,A -85,B 0,C 180,E1 -14554.888,E2 -14554.888} C_VEL
LIN {X 0,Y 350.688,Z 383.455,A -85,B 0,C 180,E1 -14556.371,E2 -14556.371} C_VEL
LIN {X 0,Y 348.532,Z 393.089,A -85,B 0,C 180,E1 -14557.816,E2 -14557.816} C_VEL
LIN {X 0,Y 345.794,Z 404.001,A -85,B 0,C 180,E1 -14559.787,E2 -14559.787} C_VEL
LIN {X 0,Y 343.242,Z 413.025,A -85,B 0,C 180,E1 -14561.805,E2 -14561.805} C_VEL
LIN {X 0,Y 341.226,Z 420.309,A -85,B 0,C 180,E1 -14563.856,E2 -14563.856} C_VEL
LIN {X 0,Y 339.232,Z 426.943,A -85,B 0,C 180,E1 -14566.217,E2 -14566.217} C_VEL
LIN {X 0,Y 337.683,Z 431.636,A -85,B 0,C 180,E1 -14568.414,E2 -14568.414} C_VEL
LIN {X 0,Y 336.466,Z 434.748,A -85,B 0,C 180,E1 -14570.381,E2 -14570.381} C_VEL
LIN {X 0,Y 335.337,Z 437.256,A -85,B 0,C 180,E1 -14572.776,E2 -14572.776} C_VEL
LIN {X 0,Y 334.623,Z 438.392,A -85,B 0,C 180,E1 -14575.181,E2 -14575.181} C_VEL
LIN {X 0,Y 334.132,Z 438.196,A -85,B 0,C 180,E1 -14577.589,E2 -14577.589} C_VEL
LIN {X 0,Y 333.893,Z 436.659,A -85,B 0,C 180,E1 -14580,E2 -14580} C_VEL
LIN {X 0,Y 333.799,Z 433.782,A -85,B 0,C 180,E1 -14582.414,E2 -14582.414} C_VEL
LIN {X 0,Y 333.765,Z 430.73,A -85,B 0,C 180,E1 -14584.227,E2 -14584.227} C_VEL
LIN {X 0,Y 334.184,Z 426.772,A -85,B 0,C 180,E1 -14586.036,E2 -14586.036} C_VEL
LIN {X 0,Y 334.583,Z 421.904,A -85,B 0,C 180,E1 -14587.848,E2 -14587.848} C_VEL
LIN {X 0,Y 335.193,Z 414.963,A -85,B 0,C 180,E1 -14589.961,E2 -14589.961} C_VEL
LIN {X 0,Y 335.974,Z 406.459,A -85,B 0,C 180,E1 -14592.075,E2 -14592.075} C_VEL
LIN {X 0,Y 336.819,Z 397.655,A -85,B 0,C 180,E1 -14593.884,E2 -14593.884} C_VEL
LIN {X 0,Y 337.874,Z 387.121,A -85,B 0,C 180,E1 -14595.689,E2 -14595.689} C_VEL
LIN {X 0,Y 338.981,Z 376.483,A -85,B 0,C 180,E1 -14597.211,E2 -14597.211} C_VEL
LIN {X 0,Y 340.11,Z 364.161,A -85,B 0,C 180,E1 -14598.681,E2 -14598.681} C_VEL
LIN {X 0,Y 340.734,Z 356.244,A -85,B 0,C 180,E1 -14599.491,E2 -14599.491} C_VEL
LIN {X 0,Y 337.061,Z 343.033,A -85,B 0,C 180,E1 -14600.865,E2 -14600.865} C_VEL
LIN {X 0,Y 333.839,Z 332.248,A -85,B 0,C 180,E1 -14601.861,E2 -14601.861} C_VEL
LIN {X 0,Y 333.725,Z 331.582,A -85,B 0,C 180,E1 -14602.086,E2 -14602.086} C_VEL
LIN {X 0,Y 333.741,Z 331.536,A -85,B 0,C 180,E1 -14606.246,E2 -14606.246} C_VEL
LIN {X 0,Y 333.716,Z 331.541,A -85,B 0,C 180,E1 -14608.972,E2 -14608.972} C_VEL
LIN {X 0,Y 333.648,Z 331.552,A -85,B 0,C 180,E1 -14612.587,E2 -14612.587} C_VEL
LIN {X 0,Y 333.681,Z 331.544,A -85,B 0,C 180,E1 -14616.139,E2 -14616.139} C_VEL
LIN {X 0,Y 333.652,Z 331.546,A -85,B 0,C 180,E1 -14619.192,E2 -14619.192} C_VEL
LIN {X 0,Y 333.638,Z 331.553,A -85,B 0,C 180,E1 -14622.5,E2 -14622.5} C_VEL
LIN {X 0,Y 333.615,Z 331.552,A -85,B 0,C 180,E1 -14625.957,E2 -14625.957} C_VEL
LIN {X 0,Y 333.662,Z 331.544,A -85,B 0,C 180,E1 -14629.313,E2 -14629.313} C_VEL
LIN {X 0,Y 333.661,Z 331.55,A -85,B 0,C 180,E1 -14632.349,E2 -14632.349} C_VEL
LIN {X 0,Y 333.68,Z 331.542,A -85,B 0,C 180,E1 -14635.341,E2 -14635.341} C_VEL
LIN {X 0,Y 333.696,Z 331.541,A -85,B 0,C 180,E1 -14639.637,E2 -14639.637} C_VEL
LIN {X 0,Y 333.745,Z 331.538,A -85,B 0,C 180,E1 -14642.4,E2 -14642.4} C_VEL
LIN {X 0,Y 333.731,Z 331.536,A -85,B 0,C 180,E1 -14645.09,E2 -14645.09} C_VEL
LIN {X 0,Y 333.681,Z 331.542,A -85,B 0,C 180,E1 -14649.018,E2 -14649.018} C_VEL
LIN {X 0,Y 333.8,Z 331.529,A -85,B 0,C 180,E1 -14651.589,E2 -14651.589} C_VEL
LIN {X 0,Y 333.814,Z 331.528,A -85,B 0,C 180,E1 -14655.576,E2 -14655.576} C_VEL
LIN {X 0,Y 333.839,Z 331.522,A -85,B 0,C 180,E1 -14659.077,E2 -14659.077} C_VEL
LIN {X 0,Y 334.03,Z 331.499,A -85,B 0,C 180,E1 -14662.747,E2 -14662.747} C_VEL
LIN {X 0,Y 333.815,Z 331.526,A -85,B 0,C 180,E1 -14665.168,E2 -14665.168} C_VEL
LIN {X 0,Y 334.11,Z 331.493,A -85,B 0,C 180,E1 -14667.588,E2 -14667.588} C_VEL
LIN {X 0,Y 334.25,Z 331.474,A -85,B 0,C 180,E1 -14669.999,E2 -14669.999} C_VEL
LIN {X 0,Y 334.11,Z 331.489,A -85,B 0,C 180,E1 -14672.41,E2 -14672.41} C_VEL
LIN {X 0,Y 334.03,Z 331.501,A -85,B 0,C 180,E1 -14677.251,E2 -14677.251} C_VEL
LIN {X 0,Y 333.837,Z 331.523,A -85,B 0,C 180,E1 -14680.921,E2 -14680.921} C_VEL
LIN {X 0,Y 333.811,Z 331.526,A -85,B 0,C 180,E1 -14684.633,E2 -14684.633} C_VEL
LIN {X 0,Y 333.798,Z 331.528,A -85,B 0,C 180,E1 -14688.654,E2 -14688.654} C_VEL
LIN {X 0,Y 333.693,Z 331.54,A -85,B 0,C 180,E1 -14692.277,E2 -14692.277} C_VEL
LIN {X 0,Y 333.735,Z 331.535,A -85,B 0,C 180,E1 -14696.245,E2 -14696.245} C_VEL
LIN {X 0,Y 333.69,Z 331.544,A -85,B 0,C 180,E1 -14698.973,E2 -14698.973} C_VEL
LIN {X 0,Y 333.642,Z 331.547,A -85,B 0,C 180,E1 -14702.586,E2 -14702.586} C_VEL
LIN {X 0,Y 333.674,Z 331.543,A -85,B 0,C 180,E1 -14706.137,E2 -14706.137} C_VEL
LIN {X 0,Y 333.644,Z 331.552,A -85,B 0,C 180,E1 -14709.191,E2 -14709.191} C_VEL
LIN {X 0,Y 333.63,Z 331.549,A -85,B 0,C 180,E1 -14712.499,E2 -14712.499} C_VEL
LIN {X 0,Y 333.618,Z 331.55,A -85,B 0,C 180,E1 -14715.958,E2 -14715.958} C_VEL
LIN {X 0,Y 333.643,Z 331.55,A -85,B 0,C 180,E1 -14719.314,E2 -14719.314} C_VEL
LIN {X 0,Y 333.661,Z 331.548,A -85,B 0,C 180,E1 -14723.166,E2 -14723.166} C_VEL
LIN {X 0,Y 333.637,Z 331.553,A -85,B 0,C 180,E1 -14726.791,E2 -14726.791} C_VEL
LIN {X 0,Y 333.699,Z 331.54,A -85,B 0,C 180,E1 -14729.709,E2 -14729.709} C_VEL
LIN {X 0,Y 333.739,Z 331.537,A -85,B 0,C 180,E1 -14732.4,E2 -14732.4} C_VEL
LIN {X 0,Y 333.714,Z 331.542,A -85,B 0,C 180,E1 -14734.932,E2 -14734.932} C_VEL
LIN {X 0,Y 333.07,Z 331.62,A -85,B 0,C 180,E1 -14735.939,E2 -14735.939} C_VEL
LIN {X 0,Y 330.201,Z 331.976,A -85,B 0,C 180,E1 -14737.578,E2 -14737.578} C_VEL
LIN {X 0,Y 327.764,Z 332.283,A -85,B 0,C 180,E1 -14738.906,E2 -14738.906} C_VEL
LIN {X 0,Y 326.736,Z 332.408,A -85,B 0,C 180,E1 -14739.934,E2 -14739.934} C_VEL
LIN {X 0,Y 326.662,Z 332.415,A -85,B 0,C 180,E1 -14740.282,E2 -14740.282} C_VEL
LIN {X 0,Y 326.721,Z 332.409,A -85,B 0,C 180,E1 -14743.761,E2 -14743.761} C_VEL
LIN {X 0,Y 326.752,Z 332.408,A -85,B 0,C 180,E1 -14746.314,E2 -14746.314} C_VEL
LIN {X 0,Y 326.806,Z 332.4,A -85,B 0,C 180,E1 -14750.093,E2 -14750.093} C_VEL
LIN {X 0,Y 326.97,Z 332.383,A -85,B 0,C 180,E1 -14752.59,E2 -14752.59} C_VEL
LIN {X 0,Y 326.772,Z 332.404,A -85,B 0,C 180,E1 -14755.064,E2 -14755.064} C_VEL
LIN {X 0,Y 327.041,Z 332.369,A -85,B 0,C 180,E1 -14757.536,E2 -14757.536} C_VEL
LIN {X 0,Y 327.191,Z 332.353,A -85,B 0,C 180,E1 -14760,E2 -14760} C_VEL
LIN {X 0,Y 327.041,Z 332.374,A -85,B 0,C 180,E1 -14762.463,E2 -14762.463} C_VEL
LIN {X 0,Y 326.988,Z 332.38,A -85,B 0,C 180,E1 -14766.169,E2 -14766.169} C_VEL
LIN {X 0,Y 326.907,Z 332.388,A -85,B 0,C 180,E1 -14768.655,E2 -14768.655} C_VEL
LIN {X 0,Y 326.731,Z 332.411,A -85,B 0,C 180,E1 -14772.421,E2 -14772.421} C_VEL
LIN {X 0,Y 326.746,Z 332.406,A -85,B 0,C 180,E1 -14774.958,E2 -14774.958} C_VEL
LIN {X 0,Y 326.725,Z 332.409,A -85,B 0,C 180,E1 -14778.839,E2 -14778.839} C_VEL
LIN {X 0,Y 326.613,Z 332.423,A -85,B 0,C 180,E1 -14782.788,E2 -14782.788} C_VEL
LIN {X 0,Y 326.682,Z 332.415,A -85,B 0,C 180,E1 -14785.484,E2 -14785.484} C_VEL
LIN {X 0,Y 326.654,Z 332.42,A -85,B 0,C 180,E1 -14789.659,E2 -14789.659} C_VEL
LIN {X 0,Y 326.616,Z 332.422,A -85,B 0,C 180,E1 -14792.948,E2 -14792.948} C_VEL
LIN {X 0,Y 326.627,Z 332.425,A -85,B 0,C 180,E1 -14797.047,E2 -14797.047} C_VEL
LIN {X 0,Y 326.67,Z 332.534,A -85,B 0,C 180,E1 -14798.415,E2 -14798.415} C_VEL
LIN {X 0,Y 328.347,Z 341.179,A -85,B 0,C 180,E1 -14802.394,E2 -14802.394} C_VEL
LIN {X 0,Y 330.16,Z 350.31,A -85,B 0,C 180,E1 -14806.364,E2 -14806.364} C_VEL
LIN {X 0,Y 331.341,Z 356.361,A -85,B 0,C 180,E1 -14808.89,E2 -14808.89} C_VEL
LIN {X 0,Y 331.188,Z 360.363,A -85,B 0,C 180,E1 -14810.462,E2 -14810.462} C_VEL
LIN {X 0,Y 329.805,Z 369.878,A -85,B 0,C 180,E1 -14814.073,E2 -14814.073} C_VEL
LIN {X 0,Y 328.411,Z 381.347,A -85,B 0,C 180,E1 -14818.352,E2 -14818.352} C_VEL
LIN {X 0,Y 327.269,Z 392.623,A -85,B 0,C 180,E1 -14822.504,E2 -14822.504} C_VEL
LIN {X 0,Y 326.768,Z 399.821,A -85,B 0,C 180,E1 -14825.035,E2 -14825.035} C_VEL
LIN {X 0,Y 328.763,Z 420.643,A -85,B 0,C 180,E1 -14826.142,E2 -14826.142} C_VEL
LIN {X 0,Y 330.115,Z 435.253,A -85,B 0,C 180,E1 -14827.162,E2 -14827.162} C_VEL
LIN {X 0,Y 331.209,Z 449.065,A -85,B 0,C 180,E1 -14828.367,E2 -14828.367} C_VEL
LIN {X 0,Y 331.441,Z 455.824,A -85,B 0,C 180,E1 -14829.044,E2 -14829.044} C_VEL
LIN {X 0,Y 329.939,Z 469.138,A -85,B 0,C 180,E1 -14830.561,E2 -14830.561} C_VEL
LIN {X 0,Y 328.685,Z 480.186,A -85,B 0,C 180,E1 -14832.101,E2 -14832.101} C_VEL
LIN {X 0,Y 327.593,Z 490.367,A -85,B 0,C 180,E1 -14833.807,E2 -14833.807} C_VEL
LIN {X 0,Y 326.716,Z 499.584,A -85,B 0,C 180,E1 -14835.665,E2 -14835.665} C_VEL
LIN {X 0,Y 326.169,Z 507.376,A -85,B 0,C 180,E1 -14837.558,E2 -14837.558} C_VEL
LIN {X 0,Y 325.939,Z 513.791,A -85,B 0,C 180,E1 -14839.44,E2 -14839.44} C_VEL
LIN {X 0,Y 325.943,Z 519.045,A -85,B 0,C 180,E1 -14841.32,E2 -14841.32} C_VEL
LIN {X 0,Y 326.089,Z 522.728,A -85,B 0,C 180,E1 -14842.922,E2 -14842.922} C_VEL
LIN {X 0,Y 326.242,Z 526.476,A -85,B 0,C 180,E1 -14845.058,E2 -14845.058} C_VEL
LIN {X 0,Y 326.489,Z 529.276,A -85,B 0,C 180,E1 -14847.534,E2 -14847.534} C_VEL
LIN {X 0,Y 326.648,Z 530.091,A -85,B 0,C 180,E1 -14848.768,E2 -14848.768} C_VEL
LIN {X 0,Y 326.784,Z 530.519,A -85,B 0,C 180,E1 -14850.001,E2 -14850.001} C_VEL
LIN {X 0,Y 326.616,Z 530.515,A -85,B 0,C 180,E1 -14851.234,E2 -14851.234} C_VEL
LIN {X 0,Y 326.177,Z 529.356,A -85,B 0,C 180,E1 -14853.707,E2 -14853.707} C_VEL
LIN {X 0,Y 326.047,Z 528.225,A -85,B 0,C 180,E1 -14854.947,E2 -14854.947} C_VEL
LIN {X 0,Y 325.694,Z 524.834,A -85,B 0,C 180,E1 -14857.44,E2 -14857.44} C_VEL
LIN {X 0,Y 325.582,Z 519.949,A -85,B 0,C 180,E1 -14859.945,E2 -14859.945} C_VEL
LIN {X 0,Y 325.906,Z 513.524,A -85,B 0,C 180,E1 -14862.454,E2 -14862.454} C_VEL
LIN {X 0,Y 326.663,Z 507.025,A -85,B 0,C 180,E1 -14864.499,E2 -14864.499} C_VEL
LIN {X 0,Y 327.941,Z 498.178,A -85,B 0,C 180,E1 -14866.818,E2 -14866.818} C_VEL
LIN {X 0,Y 329.816,Z 488.266,A -85,B 0,C 180,E1 -14868.964,E2 -14868.964} C_VEL
LIN {X 0,Y 332.195,Z 476.495,A -85,B 0,C 180,E1 -14871.08,E2 -14871.08} C_VEL
LIN {X 0,Y 335.169,Z 463.589,A -85,B 0,C 180,E1 -14872.989,E2 -14872.989} C_VEL
LIN {X 0,Y 337.029,Z 449.783,A -85,B 0,C 180,E1 -14874.814,E2 -14874.814} C_VEL
LIN {X 0,Y 338.433,Z 436.182,A -85,B 0,C 180,E1 -14876.393,E2 -14876.393} C_VEL
LIN {X 0,Y 338.423,Z 421.713,A -85,B 0,C 180,E1 -14878.043,E2 -14878.043} C_VEL
LIN {X 0,Y 337.077,Z 407.212,A -85,B 0,C 180,E1 -14879.762,E2 -14879.762} C_VEL
LIN {X 0,Y 334.582,Z 392.38,A -85,B 0,C 180,E1 -14881.678,E2 -14881.678} C_VEL
LIN {X 0,Y 332.788,Z 384.733,A -85,B 0,C 180,E1 -14882.795,E2 -14882.795} C_VEL
LIN {X 0,Y 331.384,Z 379.307,A -85,B 0,C 180,E1 -14883.647,E2 -14883.647} C_VEL
LIN {X 0,Y 330.738,Z 377.107,A -85,B 0,C 180,E1 -14884.032,E2 -14884.032} C_VEL
LIN {X 0,Y 329.34,Z 371.977,A -85,B 0,C 180,E1 -14884.94,E2 -14884.94} C_VEL
LIN {X 0,Y 329.216,Z 369.704,A -85,B 0,C 180,E1 -14885.438,E2 -14885.438} C_VEL
LIN {X 0,Y 331.278,Z 360.255,A -85,B 0,C 180,E1 -14889.528,E2 -14889.528} C_VEL
LIN {X 0,Y 331.662,Z 358.618,A -85,B 0,C 180,E1 -14890.284,E2 -14890.284} C_VEL
LIN {X 0,Y 331.423,Z 355.275,A -85,B 0,C 180,E1 -14892.082,E2 -14892.082} C_VEL
LIN {X 0,Y 330.715,Z 351.266,A -85,B 0,C 180,E1 -14894.531,E2 -14894.531} C_VEL
LIN {X 0,Y 329.951,Z 347.71,A -85,B 0,C 180,E1 -14897.031,E2 -14897.031} C_VEL
LIN {X 0,Y 329.14,Z 343.868,A -85,B 0,C 180,E1 -14900.238,E2 -14900.238} C_VEL
LIN {X 0,Y 328.465,Z 340.755,A -85,B 0,C 180,E1 -14903.661,E2 -14903.661} C_VEL
LIN {X 0,Y 328.77,Z 341.218,A -85,B 0,C 180,E1 -14904.173,E2 -14904.173} C_VEL
LIN {X 0,Y 329.943,Z 342.435,A -85,B 0,C 180,E1 -14904.892,E2 -14904.892} C_VEL
LIN {X 0,Y 331.689,Z 343.265,A -85,B 0,C 180,E1 -14905.727,E2 -14905.727} C_VEL
LIN {X 0,Y 336.341,Z 348.099,A -85,B 0,C 180,E1 -14907.951,E2 -14907.951} C_VEL
LIN {X 0,Y 337.941,Z 350.053,A -85,B 0,C 180,E1 -14908.674,E2 -14908.674} C_VEL
LIN {X 0,Y 341.232,Z 356.438,A -85,B 0,C 180,E1 -14910.376,E2 -14910.376} C_VEL
LIN {X 0,Y 344.181,Z 363.276,A -85,B 0,C 180,E1 -14911.989,E2 -14911.989} C_VEL
LIN {X 0,Y 346.87,Z 372.254,A -85,B 0,C 180,E1 -14913.854,E2 -14913.854} C_VEL
LIN {X 0,Y 347.326,Z 375.475,A -85,B 0,C 180,E1 -14914.45,E2 -14914.45} C_VEL
LIN {X 0,Y 344.721,Z 386.813,A -85,B 0,C 180,E1 -14915.937,E2 -14915.937} C_VEL
LIN {X 0,Y 341.968,Z 397.961,A -85,B 0,C 180,E1 -14917.733,E2 -14917.733} C_VEL
LIN {X 0,Y 339.179,Z 407.899,A -85,B 0,C 180,E1 -14919.692,E2 -14919.692} C_VEL
LIN {X 0,Y 336.867,Z 415.307,A -85,B 0,C 180,E1 -14921.449,E2 -14921.449} C_VEL
LIN {X 0,Y 334.718,Z 422.374,A -85,B 0,C 180,E1 -14923.534,E2 -14923.534} C_VEL
LIN {X 0,Y 332.594,Z 428.808,A -85,B 0,C 180,E1 -14925.936,E2 -14925.936} C_VEL
LIN {X 0,Y 330.81,Z 433.615,A -85,B 0,C 180,E1 -14928.357,E2 -14928.357} C_VEL
LIN {X 0,Y 329.659,Z 436.3,A -85,B 0,C 180,E1 -14930.18,E2 -14930.18} C_VEL
LIN {X 0,Y 328.444,Z 438.656,A -85,B 0,C 180,E1 -14932.624,E2 -14932.624} C_VEL
LIN {X 0,Y 327.657,Z 439.633,A -85,B 0,C 180,E1 -14935.078,E2 -14935.078} C_VEL
LIN {X 0,Y 327.124,Z 439.306,A -85,B 0,C 180,E1 -14937.538,E2 -14937.538} C_VEL
LIN {X 0,Y 326.872,Z 437.641,A -85,B 0,C 180,E1 -14940,E2 -14940} C_VEL
LIN {X 0,Y 326.872,Z 436.302,A -85,B 0,C 180,E1 -14941.232,E2 -14941.232} C_VEL
LIN {X 0,Y 326.601,Z 432.636,A -85,B 0,C 180,E1 -14943.702,E2 -14943.702} C_VEL
LIN {X 0,Y 327.182,Z 427.435,A -85,B 0,C 180,E1 -14946.166,E2 -14946.166} C_VEL
LIN {X 0,Y 327.585,Z 422.442,A -85,B 0,C 180,E1 -14948.016,E2 -14948.016} C_VEL
LIN {X 0,Y 328.221,Z 415.366,A -85,B 0,C 180,E1 -14950.175,E2 -14950.175} C_VEL
LIN {X 0,Y 329.022,Z 406.695,A -85,B 0,C 180,E1 -14952.334,E2 -14952.334} C_VEL
LIN {X 0,Y 329.921,Z 397.72,A -85,B 0,C 180,E1 -14954.181,E2 -14954.181} C_VEL
LIN {X 0,Y 331.007,Z 386.974,A -85,B 0,C 180,E1 -14956.023,E2 -14956.023} C_VEL
LIN {X 0,Y 332.282,Z 375.272,A -85,B 0,C 180,E1 -14957.684,E2 -14957.684} C_VEL
LIN {X 0,Y 333.466,Z 362.155,A -85,B 0,C 180,E1 -14959.227,E2 -14959.227} C_VEL
LIN {X 0,Y 333.773,Z 357.631,A -85,B 0,C 180,E1 -14959.688,E2 -14959.688} C_VEL
LIN {X 0,Y 330.148,Z 344.382,A -85,B 0,C 180,E1 -14961.106,E2 -14961.106} C_VEL
LIN {X 0,Y 326.798,Z 333.176,A -85,B 0,C 180,E1 -14962.161,E2 -14962.161} C_VEL
LIN {X 0,Y 326.665,Z 332.46,A -85,B 0,C 180,E1 -14962.403,E2 -14962.403} C_VEL
LIN {X 0,Y 326.695,Z 332.413,A -85,B 0,C 180,E1 -14965.484,E2 -14965.484} C_VEL
LIN {X 0,Y 326.666,Z 332.416,A -85,B 0,C 180,E1 -14969.659,E2 -14969.659} C_VEL
LIN {X 0,Y 326.612,Z 332.424,A -85,B 0,C 180,E1 -14974.019,E2 -14974.019} C_VEL
LIN {X 0,Y 326.633,Z 332.421,A -85,B 0,C 180,E1 -14977.238,E2 -14977.238} C_VEL
LIN {X 0,Y 326.583,Z 332.427,A -85,B 0,C 180,E1 -14981.131,E2 -14981.131} C_VEL
LIN {X 0,Y 326.536,Z 332.435,A -85,B 0,C 180,E1 -14984.743,E2 -14984.743} C_VEL
LIN {X 0,Y 326.603,Z 332.427,A -85,B 0,C 180,E1 -14988.157,E2 -14988.157} C_VEL
LIN {X 0,Y 326.647,Z 332.418,A -85,B 0,C 180,E1 -14991.394,E2 -14991.394} C_VEL
LIN {X 0,Y 326.626,Z 332.422,A -85,B 0,C 180,E1 -14994.851,E2 -14994.851} C_VEL
LIN {X 0,Y 326.615,Z 332.422,A -85,B 0,C 180,E1 -14997.455,E2 -14997.455} C_VEL
LIN {X 0,Y 326.653,Z 332.422,A -85,B 0,C 180,E1 -15000.339,E2 -15000.339} C_VEL
LIN {X 0,Y 326.695,Z 332.414,A -85,B 0,C 180,E1 -15004.516,E2 -15004.516} C_VEL
LIN {X 0,Y 326.626,Z 332.423,A -85,B 0,C 180,E1 -15008.543,E2 -15008.543} C_VEL
LIN {X 0,Y 326.75,Z 332.406,A -85,B 0,C 180,E1 -15011.177,E2 -15011.177} C_VEL
LIN {X 0,Y 326.769,Z 332.404,A -85,B 0,C 180,E1 -15015.432,E2 -15015.432} C_VEL
LIN {X 0,Y 326.775,Z 332.402,A -85,B 0,C 180,E1 -15018.838,E2 -15018.838} C_VEL
LIN {X 0,Y 326.984,Z 332.377,A -85,B 0,C 180,E1 -15022.589,E2 -15022.589} C_VEL
LIN {X 0,Y 326.782,Z 332.402,A -85,B 0,C 180,E1 -15025.064,E2 -15025.064} C_VEL
LIN {X 0,Y 327.051,Z 332.371,A -85,B 0,C 180,E1 -15027.536,E2 -15027.536} C_VEL
LIN {X 0,Y 327.202,Z 332.352,A -85,B 0,C 180,E1 -15029.999,E2 -15029.999} C_VEL
LIN {X 0,Y 327.051,Z 332.368,A -85,B 0,C 180,E1 -15032.462,E2 -15032.462} C_VEL
LIN {X 0,Y 327,Z 332.376,A -85,B 0,C 180,E1 -15036.168,E2 -15036.168} C_VEL
LIN {X 0,Y 326.918,Z 332.384,A -85,B 0,C 180,E1 -15038.654,E2 -15038.654} C_VEL
LIN {X 0,Y 326.738,Z 332.407,A -85,B 0,C 180,E1 -15042.42,E2 -15042.42} C_VEL
LIN {X 0,Y 326.756,Z 332.406,A -85,B 0,C 180,E1 -15044.956,E2 -15044.956} C_VEL
LIN {X 0,Y 326.734,Z 332.408,A -85,B 0,C 180,E1 -15048.837,E2 -15048.837} C_VEL
LIN {X 0,Y 326.622,Z 332.422,A -85,B 0,C 180,E1 -15052.786,E2 -15052.786} C_VEL
LIN {X 0,Y 326.69,Z 332.417,A -85,B 0,C 180,E1 -15055.482,E2 -15055.482} C_VEL
LIN {X 0,Y 326.647,Z 332.421,A -85,B 0,C 180,E1 -15059.659,E2 -15059.659} C_VEL
LIN {X 0,Y 326.606,Z 332.424,A -85,B 0,C 180,E1 -15064.018,E2 -15064.018} C_VEL
LIN {X 0,Y 326.626,Z 332.426,A -85,B 0,C 180,E1 -15067.237,E2 -15067.237} C_VEL
LIN {X 0,Y 326.576,Z 332.433,A -85,B 0,C 180,E1 -15071.13,E2 -15071.13} C_VEL
LIN {X 0,Y 326.553,Z 332.433,A -85,B 0,C 180,E1 -15074.747,E2 -15074.747} C_VEL
LIN {X 0,Y 326.573,Z 332.428,A -85,B 0,C 180,E1 -15078.153,E2 -15078.153} C_VEL
LIN {X 0,Y 326.619,Z 332.424,A -85,B 0,C 180,E1 -15081.39,E2 -15081.39} C_VEL
LIN {X 0,Y 326.615,Z 332.427,A -85,B 0,C 180,E1 -15084.85,E2 -15084.85} C_VEL
LIN {X 0,Y 326.61,Z 332.424,A -85,B 0,C 180,E1 -15087.455,E2 -15087.455} C_VEL
LIN {X 0,Y 326.656,Z 332.419,A -85,B 0,C 180,E1 -15090.34,E2 -15090.34} C_VEL
LIN {X 0,Y 326.684,Z 332.417,A -85,B 0,C 180,E1 -15094.515,E2 -15094.515} C_VEL
LIN {X 0,Y 326.642,Z 332.423,A -85,B 0,C 180,E1 -15098.545,E2 -15098.545} C_VEL
LIN {X 0,Y 326.662,Z 332.415,A -85,B 0,C 180,E1 -15100.282,E2 -15100.282} C_VEL
LIN {X 0,Y 326.028,Z 332.497,A -85,B 0,C 180,E1 -15101.311,E2 -15101.311} C_VEL
LIN {X 0,Y 323.211,Z 332.849,A -85,B 0,C 180,E1 -15102.986,E2 -15102.986} C_VEL
LIN {X 0,Y 320.814,Z 333.148,A -85,B 0,C 180,E1 -15104.344,E2 -15104.344} C_VEL
LIN {X 0,Y 319.795,Z 333.272,A -85,B 0,C 180,E1 -15105.394,E2 -15105.394} C_VEL
LIN {X 0,Y 319.718,Z 333.281,A -85,B 0,C 180,E1 -15105.75,E2 -15105.75} C_VEL
LIN {X 0,Y 319.75,Z 333.278,A -85,B 0,C 180,E1 -15109.872,E2 -15109.872} C_VEL
LIN {X 0,Y 319.927,Z 333.26,A -85,B 0,C 180,E1 -15112.426,E2 -15112.426} C_VEL
LIN {X 0,Y 319.742,Z 333.28,A -85,B 0,C 180,E1 -15114.956,E2 -15114.956} C_VEL
LIN {X 0,Y 319.985,Z 333.248,A -85,B 0,C 180,E1 -15117.482,E2 -15117.482} C_VEL
LIN {X 0,Y 320.143,Z 333.231,A -85,B 0,C 180,E1 -15120,E2 -15120} C_VEL
LIN {X 0,Y 319.984,Z 333.252,A -85,B 0,C 180,E1 -15122.517,E2 -15122.517} C_VEL
LIN {X 0,Y 319.944,Z 333.259,A -85,B 0,C 180,E1 -15126.305,E2 -15126.305} C_VEL
LIN {X 0,Y 319.835,Z 333.268,A -85,B 0,C 180,E1 -15128.848,E2 -15128.848} C_VEL
LIN {X 0,Y 319.677,Z 333.288,A -85,B 0,C 180,E1 -15132.7,E2 -15132.7} C_VEL
LIN {X 0,Y 319.692,Z 333.285,A -85,B 0,C 180,E1 -15135.296,E2 -15135.296} C_VEL
LIN {X 0,Y 319.667,Z 333.288,A -85,B 0,C 180,E1 -15139.255,E2 -15139.255} C_VEL
LIN {X 0,Y 319.562,Z 333.301,A -85,B 0,C 180,E1 -15143.32,E2 -15143.32} C_VEL
LIN {X 0,Y 319.627,Z 333.297,A -85,B 0,C 180,E1 -15146.088,E2 -15146.088} C_VEL
LIN {X 0,Y 319.582,Z 333.298,A -85,B 0,C 180,E1 -15148.934,E2 -15148.934} C_VEL
LIN {X 0,Y 319.532,Z 333.31,A -85,B 0,C 180,E1 -15151.862,E2 -15151.862} C_VEL
LIN {X 0,Y 319.574,Z 333.302,A -85,B 0,C 180,E1 -15155.544,E2 -15155.544} C_VEL
LIN {X 0,Y 319.646,Z 333.441,A -85,B 0,C 180,E1 -15158.098,E2 -15158.098} C_VEL
LIN {X 0,Y 321.194,Z 341.595,A -85,B 0,C 180,E1 -15161.933,E2 -15161.933} C_VEL
LIN {X 0,Y 322.94,Z 350.487,A -85,B 0,C 180,E1 -15165.903,E2 -15165.903} C_VEL
LIN {X 0,Y 324.2,Z 356.373,A -85,B 0,C 180,E1 -15168.424,E2 -15168.424} C_VEL
LIN {X 0,Y 324.389,Z 358.893,A -85,B 0,C 180,E1 -15169.463,E2 -15169.463} C_VEL
LIN {X 0,Y 323.293,Z 366.668,A -85,B 0,C 180,E1 -15172.507,E2 -15172.507} C_VEL
LIN {X 0,Y 321.89,Z 376.951,A -85,B 0,C 180,E1 -15176.467,E2 -15176.467} C_VEL
LIN {X 0,Y 320.902,Z 385.605,A -85,B 0,C 180,E1 -15179.755,E2 -15179.755} C_VEL
LIN {X 0,Y 319.794,Z 397.691,A -85,B 0,C 180,E1 -15184.295,E2 -15184.295} C_VEL
LIN {X 0,Y 319.732,Z 399.166,A -85,B 0,C 180,E1 -15184.699,E2 -15184.699} C_VEL
LIN {X 0,Y 321.5,Z 418.333,A -85,B 0,C 180,E1 -15185.725,E2 -15185.725} C_VEL
LIN {X 0,Y 322.888,Z 433.488,A -85,B 0,C 180,E1 -15186.79,E2 -15186.79} C_VEL
LIN {X 0,Y 324.092,Z 447.569,A -85,B 0,C 180,E1 -15188.035,E2 -15188.035} C_VEL
LIN {X 0,Y 324.325,Z 456.747,A -85,B 0,C 180,E1 -15188.986,E2 -15188.986} C_VEL
LIN {X 0,Y 322.865,Z 469.028,A -85,B 0,C 180,E1 -15190.448,E2 -15190.448} C_VEL
LIN {X 0,Y 321.628,Z 479.921,A -85,B 0,C 180,E1 -15192.023,E2 -15192.023} C_VEL
LIN {X 0,Y 320.524,Z 489.952,A -85,B 0,C 180,E1 -15193.767,E2 -15193.767} C_VEL
LIN {X 0,Y 319.621,Z 499.352,A -85,B 0,C 180,E1 -15195.742,E2 -15195.742} C_VEL
LIN {X 0,Y 319.094,Z 507.86,A -85,B 0,C 180,E1 -15197.924,E2 -15197.924} C_VEL
LIN {X 0,Y 318.875,Z 514.004,A -85,B 0,C 180,E1 -15199.846,E2 -15199.846} C_VEL
LIN {X 0,Y 318.949,Z 519.048,A -85,B 0,C 180,E1 -15201.767,E2 -15201.767} C_VEL
LIN {X 0,Y 319.139,Z 522.993,A -85,B 0,C 180,E1 -15203.68,E2 -15203.68} C_VEL
LIN {X 0,Y 319.225,Z 525.084,A -85,B 0,C 180,E1 -15204.949,E2 -15204.949} C_VEL
LIN {X 0,Y 319.482,Z 528.015,A -85,B 0,C 180,E1 -15207.48,E2 -15207.48} C_VEL
LIN {X 0,Y 319.642,Z 528.876,A -85,B 0,C 180,E1 -15208.741,E2 -15208.741} C_VEL
LIN {X 0,Y 319.777,Z 529.345,A -85,B 0,C 180,E1 -15210.001,E2 -15210.001} C_VEL
LIN {X 0,Y 319.602,Z 529.382,A -85,B 0,C 180,E1 -15211.261,E2 -15211.261} C_VEL
LIN {X 0,Y 319.124,Z 528.301,A -85,B 0,C 180,E1 -15213.789,E2 -15213.789} C_VEL
LIN {X 0,Y 318.979,Z 527.213,A -85,B 0,C 180,E1 -15215.057,E2 -15215.057} C_VEL
LIN {X 0,Y 318.612,Z 523.912,A -85,B 0,C 180,E1 -15217.606,E2 -15217.606} C_VEL
LIN {X 0,Y 318.503,Z 519.132,A -85,B 0,C 180,E1 -15220.169,E2 -15220.169} C_VEL
LIN {X 0,Y 318.872,Z 512.838,A -85,B 0,C 180,E1 -15222.734,E2 -15222.734} C_VEL
LIN {X 0,Y 319.759,Z 506.021,A -85,B 0,C 180,E1 -15224.964,E2 -15224.964} C_VEL
LIN {X 0,Y 321.336,Z 496.582,A -85,B 0,C 180,E1 -15227.502,E2 -15227.502} C_VEL
LIN {X 0,Y 323.392,Z 486.691,A -85,B 0,C 180,E1 -15229.686,E2 -15229.686} C_VEL
LIN {X 0,Y 325.914,Z 475.301,A -85,B 0,C 180,E1 -15231.781,E2 -15231.781} C_VEL
LIN {X 0,Y 329.126,Z 462.19,A -85,B 0,C 180,E1 -15233.77,E2 -15233.77} C_VEL
LIN {X 0,Y 331.217,Z 447.403,A -85,B 0,C 180,E1 -15235.785,E2 -15235.785} C_VEL
LIN {X 0,Y 332.503,Z 435.429,A -85,B 0,C 180,E1 -15237.237,E2 -15237.237} C_VEL
LIN {X 0,Y 332.577,Z 421.015,A -85,B 0,C 180,E1 -15238.999,E2 -15238.999} C_VEL
LIN {X 0,Y 331.394,Z 407.519,A -85,B 0,C 180,E1 -15240.737,E2 -15240.737} C_VEL
LIN {X 0,Y 329.666,Z 395.628,A -85,B 0,C 180,E1 -15242.392,E2 -15242.392} C_VEL
LIN {X 0,Y 328.387,Z 388.971,A -85,B 0,C 180,E1 -15243.42,E2 -15243.42} C_VEL
LIN {X 0,Y 327.354,Z 384.805,A -85,B 0,C 180,E1 -15244.136,E2 -15244.136} C_VEL
LIN {X 0,Y 327.127,Z 382.958,A -85,B 0,C 180,E1 -15244.403,E2 -15244.403} C_VEL
LIN {X 0,Y 325.717,Z 377.916,A -85,B 0,C 180,E1 -15245.386,E2 -15245.386} C_VEL
LIN {X 0,Y 325.277,Z 375.198,A -85,B 0,C 180,E1 -15245.841,E2 -15245.841} C_VEL
LIN {X 0,Y 323.643,Z 369.361,A -85,B 0,C 180,E1 -15247.149,E2 -15247.149} C_VEL
LIN {X 0,Y 323.385,Z 366.28,A -85,B 0,C 180,E1 -15247.777,E2 -15247.777} C_VEL
LIN {X 0,Y 324.024,Z 363.367,A -85,B 0,C 180,E1 -15248.978,E2 -15248.978} C_VEL
LIN {X 0,Y 324.843,Z 359.616,A -85,B 0,C 180,E1 -15250.78,E2 -15250.78} C_VEL
LIN {X 0,Y 324.269,Z 355.163,A -85,B 0,C 180,E1 -15253.361,E2 -15253.361} C_VEL
LIN {X 0,Y 323.289,Z 350.177,A -85,B 0,C 180,E1 -15256.782,E2 -15256.782} C_VEL
LIN {X 0,Y 322.302,Z 345.662,A -85,B 0,C 180,E1 -15260.708,E2 -15260.708} C_VEL
LIN {X 0,Y 322.468,Z 345.789,A -85,B 0,C 180,E1 -15261.353,E2 -15261.353} C_VEL
LIN {X 0,Y 323.803,Z 346.815,A -85,B 0,C 180,E1 -15262.575,E2 -15262.575} C_VEL
LIN {X 0,Y 324.76,Z 347.098,A -85,B 0,C 180,E1 -15263.198,E2 -15263.198} C_VEL
LIN {X 0,Y 328.249,Z 349.476,A -85,B 0,C 180,E1 -15265.315,E2 -15265.315} C_VEL
LIN {X 0,Y 332.733,Z 353.981,A -85,B 0,C 180,E1 -15267.661,E2 -15267.661} C_VEL
LIN {X 0,Y 334.58,Z 356.579,A -85,B 0,C 180,E1 -15268.627,E2 -15268.627} C_VEL
LIN {X 0,Y 337.541,Z 363.131,A -85,B 0,C 180,E1 -15270.42,E2 -15270.42} C_VEL
LIN {X 0,Y 340.234,Z 370.769,A -85,B 0,C 180,E1 -15272.246,E2 -15272.246} C_VEL
LIN {X 0,Y 341.826,Z 377.839,A -85,B 0,C 180,E1 -15273.768,E2 -15273.768} C_VEL
LIN {X 0,Y 338.829,Z 390.236,A -85,B 0,C 180,E1 -15275.491,E2 -15275.491} C_VEL
LIN {X 0,Y 336.108,Z 400.197,A -85,B 0,C 180,E1 -15277.178,E2 -15277.178} C_VEL
LIN {X 0,Y 333.359,Z 409.198,A -85,B 0,C 180,E1 -15278.998,E2 -15278.998} C_VEL
LIN {X 0,Y 330.515,Z 417.661,A -85,B 0,C 180,E1 -15281.079,E2 -15281.079} C_VEL
LIN {X 0,Y 328.244,Z 424.492,A -85,B 0,C 180,E1 -15283.199,E2 -15283.199} C_VEL
LIN {X 0,Y 326.439,Z 429.28,A -85,B 0,C 180,E1 -15285.028,E2 -15285.028} C_VEL
LIN {X 0,Y 324.464,Z 434.302,A -85,B 0,C 180,E1 -15287.491,E2 -15287.491} C_VEL
LIN {X 0,Y 322.847,Z 437.862,A -85,B 0,C 180,E1 -15289.971,E2 -15289.971} C_VEL
LIN {X 0,Y 321.564,Z 440.037,A -85,B 0,C 180,E1 -15292.465,E2 -15292.465} C_VEL
LIN {X 0,Y 320.69,Z 440.88,A -85,B 0,C 180,E1 -15294.971,E2 -15294.971} C_VEL
LIN {X 0,Y 320.116,Z 440.414,A -85,B 0,C 180,E1 -15297.484,E2 -15297.484} C_VEL
LIN {X 0,Y 319.85,Z 438.616,A -85,B 0,C 180,E1 -15300,E2 -15300} C_VEL
LIN {X 0,Y 319.851,Z 437.21,A -85,B 0,C 180,E1 -15301.259,E2 -15301.259} C_VEL
LIN {X 0,Y 319.56,Z 433.414,A -85,B 0,C 180,E1 -15303.783,E2 -15303.783} C_VEL
LIN {X 0,Y 320.159,Z 428.033,A -85,B 0,C 180,E1 -15306.302,E2 -15306.302} C_VEL
LIN {X 0,Y 320.699,Z 421.015,A -85,B 0,C 180,E1 -15308.825,E2 -15308.825} C_VEL
LIN {X 0,Y 321.397,Z 413.349,A -85,B 0,C 180,E1 -15311.031,E2 -15311.031} C_VEL
LIN {X 0,Y 322.426,Z 403.996,A -85,B 0,C 180,E1 -15313.231,E2 -15313.231} C_VEL
LIN {X 0,Y 323.355,Z 394.293,A -85,B 0,C 180,E1 -15315.119,E2 -15315.119} C_VEL
LIN {X 0,Y 324.672,Z 382.625,A -85,B 0,C 180,E1 -15316.992,E2 -15316.992} C_VEL
LIN {X 0,Y 325.932,Z 369.774,A -85,B 0,C 180,E1 -15318.698,E2 -15318.698} C_VEL
LIN {X 0,Y 326.768,Z 359.849,A -85,B 0,C 180,E1 -15319.801,E2 -15319.801} C_VEL
LIN {X 0,Y 326.286,Z 356.698,A -85,B 0,C 180,E1 -15320.16,E2 -15320.16} C_VEL
LIN {X 0,Y 322.492,Z 343.422,A -85,B 0,C 180,E1 -15321.572,E2 -15321.572} C_VEL
LIN {X 0,Y 319.696,Z 333.826,A -85,B 0,C 180,E1 -15322.514,E2 -15322.514} C_VEL
LIN {X 0,Y 319.599,Z 333.358,A -85,B 0,C 180,E1 -15322.691,E2 -15322.691} C_VEL
LIN {X 0,Y 319.64,Z 333.292,A -85,B 0,C 180,E1 -15326.088,E2 -15326.088} C_VEL
LIN {X 0,Y 319.595,Z 333.3,A -85,B 0,C 180,E1 -15328.934,E2 -15328.934} C_VEL
LIN {X 0,Y 319.537,Z 333.304,A -85,B 0,C 180,E1 -15331.862,E2 -15331.862} C_VEL
LIN {X 0,Y 319.585,Z 333.298,A -85,B 0,C 180,E1 -15335.543,E2 -15335.543} C_VEL
LIN {X 0,Y 319.562,Z 333.302,A -85,B 0,C 180,E1 -15338.01,E2 -15338.01} C_VEL
LIN {X 0,Y 319.531,Z 333.305,A -85,B 0,C 180,E1 -15341.597,E2 -15341.597} C_VEL
LIN {X 0,Y 319.499,Z 333.309,A -85,B 0,C 180,E1 -15345.258,E2 -15345.258} C_VEL
LIN {X 0,Y 319.574,Z 333.305,A -85,B 0,C 180,E1 -15348.394,E2 -15348.394} C_VEL
LIN {X 0,Y 319.603,Z 333.301,A -85,B 0,C 180,E1 -15352.339,E2 -15352.339} C_VEL
LIN {X 0,Y 319.566,Z 333.3,A -85,B 0,C 180,E1 -15355.123,E2 -15355.123} C_VEL
LIN {X 0,Y 319.572,Z 333.3,A -85,B 0,C 180,E1 -15359.059,E2 -15359.059} C_VEL
LIN {X 0,Y 319.611,Z 333.297,A -85,B 0,C 180,E1 -15362.497,E2 -15362.497} C_VEL
LIN {X 0,Y 319.608,Z 333.295,A -85,B 0,C 180,E1 -15365.303,E2 -15365.303} C_VEL
LIN {X 0,Y 319.609,Z 333.296,A -85,B 0,C 180,E1 -15369.4,E2 -15369.4} C_VEL
LIN {X 0,Y 319.664,Z 333.293,A -85,B 0,C 180,E1 -15372.072,E2 -15372.072} C_VEL
LIN {X 0,Y 319.738,Z 333.284,A -85,B 0,C 180,E1 -15376.007,E2 -15376.007} C_VEL
LIN {X 0,Y 319.763,Z 333.281,A -85,B 0,C 180,E1 -15379.872,E2 -15379.872} C_VEL
LIN {X 0,Y 319.938,Z 333.255,A -85,B 0,C 180,E1 -15382.425,E2 -15382.425} C_VEL
LIN {X 0,Y 319.751,Z 333.277,A -85,B 0,C 180,E1 -15384.955,E2 -15384.955} C_VEL
LIN {X 0,Y 319.994,Z 333.25,A -85,B 0,C 180,E1 -15387.481,E2 -15387.481} C_VEL
LIN {X 0,Y 320.154,Z 333.23,A -85,B 0,C 180,E1 -15389.999,E2 -15389.999} C_VEL
LIN {X 0,Y 319.994,Z 333.247,A -85,B 0,C 180,E1 -15392.516,E2 -15392.516} C_VEL
LIN {X 0,Y 319.956,Z 333.252,A -85,B 0,C 180,E1 -15396.304,E2 -15396.304} C_VEL
LIN {X 0,Y 319.846,Z 333.266,A -85,B 0,C 180,E1 -15398.847,E2 -15398.847} C_VEL
LIN {X 0,Y 319.685,Z 333.286,A -85,B 0,C 180,E1 -15402.698,E2 -15402.698} C_VEL
LIN {X 0,Y 319.702,Z 333.287,A -85,B 0,C 180,E1 -15405.294,E2 -15405.294} C_VEL
LIN {X 0,Y 319.676,Z 333.29,A -85,B 0,C 180,E1 -15409.254,E2 -15409.254} C_VEL
LIN {X 0,Y 319.571,Z 333.305,A -85,B 0,C 180,E1 -15413.318,E2 -15413.318} C_VEL
LIN {X 0,Y 319.618,Z 333.294,A -85,B 0,C 180,E1 -15416.088,E2 -15416.088} C_VEL
LIN {X 0,Y 319.58,Z 333.301,A -85,B 0,C 180,E1 -15418.933,E2 -15418.933} C_VEL
LIN {X 0,Y 319.53,Z 333.306,A -85,B 0,C 180,E1 -15421.86,E2 -15421.86} C_VEL
LIN {X 0,Y 319.578,Z 333.301,A -85,B 0,C 180,E1 -15425.542,E2 -15425.542} C_VEL
LIN {X 0,Y 319.556,Z 333.303,A -85,B 0,C 180,E1 -15429.667,E2 -15429.667} C_VEL
LIN {X 0,Y 319.554,Z 333.304,A -85,B 0,C 180,E1 -15433.466,E2 -15433.466} C_VEL
LIN {X 0,Y 319.557,Z 333.307,A -85,B 0,C 180,E1 -15437.016,E2 -15437.016} C_VEL
LIN {X 0,Y 319.543,Z 333.304,A -85,B 0,C 180,E1 -15440.37,E2 -15440.37} C_VEL
LIN {X 0,Y 319.554,Z 333.303,A -85,B 0,C 180,E1 -15443.571,E2 -15443.571} C_VEL
LIN {X 0,Y 319.573,Z 333.303,A -85,B 0,C 180,E1 -15446.685,E2 -15446.685} C_VEL
LIN {X 0,Y 319.588,Z 333.298,A -85,B 0,C 180,E1 -15449.616,E2 -15449.616} C_VEL
LIN {X 0,Y 319.604,Z 333.299,A -85,B 0,C 180,E1 -15452.497,E2 -15452.497} C_VEL
LIN {X 0,Y 319.599,Z 333.297,A -85,B 0,C 180,E1 -15455.303,E2 -15455.303} C_VEL
LIN {X 0,Y 319.591,Z 333.298,A -85,B 0,C 180,E1 -15458.047,E2 -15458.047} C_VEL
LIN {X 0,Y 319.682,Z 333.289,A -85,B 0,C 180,E1 -15460.961,E2 -15460.961} C_VEL
LIN {X 0,Y 319.724,Z 333.281,A -85,B 0,C 180,E1 -15465.275,E2 -15465.275} C_VEL
LIN {X 0,Y 319.718,Z 333.281,A -85,B 0,C 180,E1 -15465.75,E2 -15465.75} C_VEL
LIN {X 0,Y 319.081,Z 333.365,A -85,B 0,C 180,E1 -15466.801,E2 -15466.801} C_VEL
LIN {X 0,Y 316.293,Z 333.713,A -85,B 0,C 180,E1 -15468.513,E2 -15468.513} C_VEL
LIN {X 0,Y 313.922,Z 334.007,A -85,B 0,C 180,E1 -15469.9,E2 -15469.9} C_VEL
LIN {X 0,Y 312.908,Z 334.132,A -85,B 0,C 180,E1 -15470.973,E2 -15470.973} C_VEL
LIN {X 0,Y 312.828,Z 334.14,A -85,B 0,C 180,E1 -15471.336,E2 -15471.336} C_VEL
LIN {X 0,Y 312.903,Z 334.13,A -85,B 0,C 180,E1 -15473.552,E2 -15473.552} C_VEL
LIN {X 0,Y 312.931,Z 334.127,A -85,B 0,C 180,E1 -15477.425,E2 -15477.425} C_VEL
LIN {X 0,Y 313.095,Z 334.109,A -85,B 0,C 180,E1 -15480,E2 -15480} C_VEL
LIN {X 0,Y 312.931,Z 334.13,A -85,B 0,C 180,E1 -15482.574,E2 -15482.574} C_VEL
LIN {X 0,Y 312.902,Z 334.134,A -85,B 0,C 180,E1 -15486.448,E2 -15486.448} C_VEL
LIN {X 0,Y 312.78,Z 334.146,A -85,B 0,C 180,E1 -15489.049,E2 -15489.049} C_VEL
LIN {X 0,Y 312.629,Z 334.165,A -85,B 0,C 180,E1 -15492.991,E2 -15492.991} C_VEL
LIN {X 0,Y 312.631,Z 334.166,A -85,B 0,C 180,E1 -15495.65,E2 -15495.65} C_VEL
LIN {X 0,Y 312.623,Z 334.165,A -85,B 0,C 180,E1 -15499.237,E2 -15499.237} C_VEL
LIN {X 0,Y 312.538,Z 334.176,A -85,B 0,C 180,E1 -15502.79,E2 -15502.79} C_VEL
LIN {X 0,Y 312.595,Z 334.174,A -85,B 0,C 180,E1 -15505.936,E2 -15505.936} C_VEL
LIN {X 0,Y 312.539,Z 334.178,A -85,B 0,C 180,E1 -15509.65,E2 -15509.65} C_VEL
LIN {X 0,Y 312.513,Z 334.183,A -85,B 0,C 180,E1 -15513.69,E2 -15513.69} C_VEL
LIN {X 0,Y 312.595,Z 334.328,A -85,B 0,C 180,E1 -15517.764,E2 -15517.764} C_VEL
LIN {X 0,Y 313.988,Z 341.7,A -85,B 0,C 180,E1 -15521.322,E2 -15521.322} C_VEL
LIN {X 0,Y 315.739,Z 350.633,A -85,B 0,C 180,E1 -15525.421,E2 -15525.421} C_VEL
LIN {X 0,Y 317.314,Z 358.489,A -85,B 0,C 180,E1 -15528.855,E2 -15528.855} C_VEL
LIN {X 0,Y 316.877,Z 363.555,A -85,B 0,C 180,E1 -15530.919,E2 -15530.919} C_VEL
LIN {X 0,Y 315.43,Z 372.84,A -85,B 0,C 180,E1 -15534.601,E2 -15534.601} C_VEL
LIN {X 0,Y 314.046,Z 384.133,A -85,B 0,C 180,E1 -15539.023,E2 -15539.023} C_VEL
LIN {X 0,Y 312.928,Z 395.244,A -85,B 0,C 180,E1 -15543.311,E2 -15543.311} C_VEL
LIN {X 0,Y 312.71,Z 398.111,A -85,B 0,C 180,E1 -15544.313,E2 -15544.313} C_VEL
LIN {X 0,Y 314.523,Z 418.386,A -85,B 0,C 180,E1 -15545.448,E2 -15545.448} C_VEL
LIN {X 0,Y 315.879,Z 433.66,A -85,B 0,C 180,E1 -15546.567,E2 -15546.567} C_VEL
LIN {X 0,Y 317.008,Z 447.637,A -85,B 0,C 180,E1 -15547.86,E2 -15547.86} C_VEL
LIN {X 0,Y 317.322,Z 456.333,A -85,B 0,C 180,E1 -15548.795,E2 -15548.795} C_VEL
LIN {X 0,Y 315.8,Z 468.819,A -85,B 0,C 180,E1 -15550.331,E2 -15550.331} C_VEL
LIN {X 0,Y 314.445,Z 480.506,A -85,B 0,C 180,E1 -15552.104,E2 -15552.104} C_VEL
LIN {X 0,Y 313.287,Z 491.055,A -85,B 0,C 180,E1 -15554.051,E2 -15554.051} C_VEL
LIN {X 0,Y 312.471,Z 499.834,A -85,B 0,C 180,E1 -15556.009,E2 -15556.009} C_VEL
LIN {X 0,Y 312.005,Z 508.279,A -85,B 0,C 180,E1 -15558.305,E2 -15558.305} C_VEL
LIN {X 0,Y 311.853,Z 514.133,A -85,B 0,C 180,E1 -15560.27,E2 -15560.27} C_VEL
LIN {X 0,Y 312.03,Z 520.044,A -85,B 0,C 180,E1 -15562.769,E2 -15562.769} C_VEL
LIN {X 0,Y 312.216,Z 523.647,A -85,B 0,C 180,E1 -15564.835,E2 -15564.835} C_VEL
LIN {X 0,Y 312.472,Z 526.696,A -85,B 0,C 180,E1 -15567.423,E2 -15567.423} C_VEL
LIN {X 0,Y 312.636,Z 527.622,A -85,B 0,C 180,E1 -15568.713,E2 -15568.713} C_VEL
LIN {X 0,Y 312.791,Z 528.155,A -85,B 0,C 180,E1 -15570.001,E2 -15570.001} C_VEL
LIN {X 0,Y 312.585,Z 528.238,A -85,B 0,C 180,E1 -15571.289,E2 -15571.289} C_VEL
LIN {X 0,Y 312.071,Z 527.248,A -85,B 0,C 180,E1 -15573.875,E2 -15573.875} C_VEL
LIN {X 0,Y 311.914,Z 526.206,A -85,B 0,C 180,E1 -15575.172,E2 -15575.172} C_VEL
LIN {X 0,Y 311.521,Z 523,A -85,B 0,C 180,E1 -15577.781,E2 -15577.781} C_VEL
LIN {X 0,Y 311.444,Z 518.34,A -85,B 0,C 180,E1 -15580.402,E2 -15580.402} C_VEL
LIN {X 0,Y 311.843,Z 512.186,A -85,B 0,C 180,E1 -15583.026,E2 -15583.026} C_VEL
LIN {X 0,Y 312.768,Z 505.821,A -85,B 0,C 180,E1 -15585.218,E2 -15585.218} C_VEL
LIN {X 0,Y 314.247,Z 497.568,A -85,B 0,C 180,E1 -15587.574,E2 -15587.574} C_VEL
LIN {X 0,Y 316.335,Z 488.157,A -85,B 0,C 180,E1 -15589.805,E2 -15589.805} C_VEL
LIN {X 0,Y 318.992,Z 477.098,A -85,B 0,C 180,E1 -15591.997,E2 -15591.997} C_VEL
LIN {X 0,Y 322.468,Z 464.079,A -85,B 0,C 180,E1 -15594.121,E2 -15594.121} C_VEL
LIN {X 0,Y 324.77,Z 450.014,A -85,B 0,C 180,E1 -15596.163,E2 -15596.163} C_VEL
LIN {X 0,Y 326.409,Z 438.208,A -85,B 0,C 180,E1 -15597.692,E2 -15597.692} C_VEL
LIN {X 0,Y 326.907,Z 424.884,A -85,B 0,C 180,E1 -15599.427,E2 -15599.427} C_VEL
LIN {X 0,Y 326.237,Z 411.324,A -85,B 0,C 180,E1 -15601.277,E2 -15601.277} C_VEL
LIN {X 0,Y 325.026,Z 400.351,A -85,B 0,C 180,E1 -15602.888,E2 -15602.888} C_VEL
LIN {X 0,Y 323.791,Z 392.718,A -85,B 0,C 180,E1 -15604.144,E2 -15604.144} C_VEL
LIN {X 0,Y 322.95,Z 387.486,A -85,B 0,C 180,E1 -15605.045,E2 -15605.045} C_VEL
LIN {X 0,Y 321.744,Z 381.983,A -85,B 0,C 180,E1 -15606.142,E2 -15606.142} C_VEL
LIN {X 0,Y 321.471,Z 379.926,A -85,B 0,C 180,E1 -15606.518,E2 -15606.518} C_VEL
LIN {X 0,Y 320.121,Z 373.704,A -85,B 0,C 180,E1 -15607.932,E2 -15607.932} C_VEL
LIN {X 0,Y 319.794,Z 371.055,A -85,B 0,C 180,E1 -15608.482,E2 -15608.482} C_VEL
LIN {X 0,Y 318.245,Z 361.832,A -85,B 0,C 180,E1 -15611.097,E2 -15611.097} C_VEL
LIN {X 0,Y 317.84,Z 359.132,A -85,B 0,C 180,E1 -15612.308,E2 -15612.308} C_VEL
LIN {X 0,Y 317.14,Z 355.211,A -85,B 0,C 180,E1 -15614.835,E2 -15614.835} C_VEL
LIN {X 0,Y 316.968,Z 353.571,A -85,B 0,C 180,E1 -15616.58,E2 -15616.58} C_VEL
LIN {X 0,Y 317.705,Z 352.842,A -85,B 0,C 180,E1 -15618.775,E2 -15618.775} C_VEL
LIN {X 0,Y 319.133,Z 352.274,A -85,B 0,C 180,E1 -15620.425,E2 -15620.425} C_VEL
LIN {X 0,Y 322.864,Z 354.207,A -85,B 0,C 180,E1 -15623.65,E2 -15623.65} C_VEL
LIN {X 0,Y 325.267,Z 355.896,A -85,B 0,C 180,E1 -15625.192,E2 -15625.192} C_VEL
LIN {X 0,Y 328.824,Z 359.575,A -85,B 0,C 180,E1 -15627.267,E2 -15627.267} C_VEL
LIN {X 0,Y 330.542,Z 362.026,A -85,B 0,C 180,E1 -15628.265,E2 -15628.265} C_VEL
LIN {X 0,Y 333.448,Z 369.262,A -85,B 0,C 180,E1 -15630.349,E2 -15630.349} C_VEL
LIN {X 0,Y 335.465,Z 376.254,A -85,B 0,C 180,E1 -15632.089,E2 -15632.089} C_VEL
LIN {X 0,Y 336.347,Z 381.587,A -85,B 0,C 180,E1 -15633.27,E2 -15633.27} C_VEL
LIN {X 0,Y 333.506,Z 391.874,A -85,B 0,C 180,E1 -15634.74,E2 -15634.74} C_VEL
LIN {X 0,Y 330.249,Z 402.717,A -85,B 0,C 180,E1 -15636.637,E2 -15636.637} C_VEL
LIN {X 0,Y 327.209,Z 411.897,A -85,B 0,C 180,E1 -15638.584,E2 -15638.584} C_VEL
LIN {X 0,Y 324.219,Z 420.07,A -85,B 0,C 180,E1 -15640.697,E2 -15640.697} C_VEL
LIN {X 0,Y 321.785,Z 426.641,A -85,B 0,C 180,E1 -15642.852,E2 -15642.852} C_VEL
LIN {X 0,Y 319.343,Z 432.573,A -85,B 0,C 180,E1 -15645.341,E2 -15645.341} C_VEL
LIN {X 0,Y 317.766,Z 436.065,A -85,B 0,C 180,E1 -15647.223,E2 -15647.223} C_VEL
LIN {X 0,Y 316.034,Z 439.418,A -85,B 0,C 180,E1 -15649.753,E2 -15649.753} C_VEL
LIN {X 0,Y 314.679,Z 441.432,A -85,B 0,C 180,E1 -15652.299,E2 -15652.299} C_VEL
LIN {X 0,Y 313.725,Z 442.133,A -85,B 0,C 180,E1 -15654.859,E2 -15654.859} C_VEL
LIN {X 0,Y 313.108,Z 441.52,A -85,B 0,C 180,E1 -15657.427,E2 -15657.427} C_VEL
LIN {X 0,Y 312.828,Z 439.582,A -85,B 0,C 180,E1 -15660,E2 -15660} C_VEL
LIN {X 0,Y 312.829,Z 438.106,A -85,B 0,C 180,E1 -15661.288,E2 -15661.288} C_VEL
LIN {X 0,Y 312.604,Z 435.245,A -85,B 0,C 180,E1 -15663.222,E2 -15663.222} C_VEL
LIN {X 0,Y 312.77,Z 431.567,A -85,B 0,C 180,E1 -15665.157,E2 -15665.157} C_VEL
LIN {X 0,Y 313.359,Z 425.641,A -85,B 0,C 180,E1 -15667.582,E2 -15667.582} C_VEL
LIN {X 0,Y 313.972,Z 418.348,A -85,B 0,C 180,E1 -15669.964,E2 -15669.964} C_VEL
LIN {X 0,Y 314.838,Z 409.729,A -85,B 0,C 180,E1 -15672.244,E2 -15672.244} C_VEL
LIN {X 0,Y 315.739,Z 400.923,A -85,B 0,C 180,E1 -15674.173,E2 -15674.173} C_VEL
LIN {X 0,Y 316.854,Z 390.437,A -85,B 0,C 180,E1 -15676.097,E2 -15676.097} C_VEL
LIN {X 0,Y 318.144,Z 378.898,A -85,B 0,C 180,E1 -15677.849,E2 -15677.849} C_VEL
LIN {X 0,Y 319.387,Z 366.28,A -85,B 0,C 180,E1 -15679.44,E2 -15679.44} C_VEL
LIN {X 0,Y 319.856,Z 360.457,A -85,B 0,C 180,E1 -15680.08,E2 -15680.08} C_VEL
LIN {X 0,Y 316.912,Z 349.359,A -85,B 0,C 180,E1 -15681.342,E2 -15681.342} C_VEL
LIN {X 0,Y 312.639,Z 334.717,A -85,B 0,C 180,E1 -15682.828,E2 -15682.828} C_VEL
LIN {X 0,Y 312.542,Z 334.222,A -85,B 0,C 180,E1 -15683.03,E2 -15683.03} C_VEL
LIN {X 0,Y 312.588,Z 334.175,A -85,B 0,C 180,E1 -15686.723,E2 -15686.723} C_VEL
LIN {X 0,Y 312.551,Z 334.174,A -85,B 0,C 180,E1 -15689.65,E2 -15689.65} C_VEL
LIN {X 0,Y 312.525,Z 334.178,A -85,B 0,C 180,E1 -15693.689,E2 -15693.689} C_VEL
LIN {X 0,Y 312.531,Z 334.177,A -85,B 0,C 180,E1 -15697.385,E2 -15697.385} C_VEL
LIN {X 0,Y 312.495,Z 334.185,A -85,B 0,C 180,E1 -15700.709,E2 -15700.709} C_VEL
LIN {X 0,Y 312.459,Z 334.189,A -85,B 0,C 180,E1 -15704.209,E2 -15704.209} C_VEL
LIN {X 0,Y 312.533,Z 334.178,A -85,B 0,C 180,E1 -15707.91,E2 -15707.91} C_VEL
LIN {X 0,Y 312.548,Z 334.176,A -85,B 0,C 180,E1 -15711.908,E2 -15711.908} C_VEL
LIN {X 0,Y 312.512,Z 334.181,A -85,B 0,C 180,E1 -15715.79,E2 -15715.79} C_VEL
LIN {X 0,Y 312.526,Z 334.178,A -85,B 0,C 180,E1 -15718.853,E2 -15718.853} C_VEL
LIN {X 0,Y 312.576,Z 334.173,A -85,B 0,C 180,E1 -15721.824,E2 -15721.824} C_VEL
LIN {X 0,Y 312.59,Z 334.17,A -85,B 0,C 180,E1 -15724.71,E2 -15724.71} C_VEL
LIN {X 0,Y 312.544,Z 334.175,A -85,B 0,C 180,E1 -15728.912,E2 -15728.912} C_VEL
LIN {X 0,Y 312.644,Z 334.165,A -85,B 0,C 180,E1 -15731.656,E2 -15731.656} C_VEL
LIN {X 0,Y 312.699,Z 334.159,A -85,B 0,C 180,E1 -15735.685,E2 -15735.685} C_VEL
LIN {X 0,Y 312.707,Z 334.158,A -85,B 0,C 180,E1 -15739.641,E2 -15739.641} C_VEL
LIN {X 0,Y 312.877,Z 334.136,A -85,B 0,C 180,E1 -15742.253,E2 -15742.253} C_VEL
LIN {X 0,Y 312.722,Z 334.153,A -85,B 0,C 180,E1 -15744.841,E2 -15744.841} C_VEL
LIN {X 0,Y 312.993,Z 334.119,A -85,B 0,C 180,E1 -15748.712,E2 -15748.712} C_VEL
LIN {X 0,Y 312.993,Z 334.121,A -85,B 0,C 180,E1 -15751.285,E2 -15751.285} C_VEL
LIN {X 0,Y 312.722,Z 334.154,A -85,B 0,C 180,E1 -15755.156,E2 -15755.156} C_VEL
LIN {X 0,Y 312.876,Z 334.138,A -85,B 0,C 180,E1 -15757.744,E2 -15757.744} C_VEL
LIN {X 0,Y 312.672,Z 334.164,A -85,B 0,C 180,E1 -15761.67,E2 -15761.67} C_VEL
LIN {X 0,Y 312.702,Z 334.156,A -85,B 0,C 180,E1 -15764.886,E2 -15764.886} C_VEL
LIN {X 0,Y 312.632,Z 334.168,A -85,B 0,C 180,E1 -15769.235,E2 -15769.235} C_VEL
LIN {X 0,Y 312.547,Z 334.175,A -85,B 0,C 180,E1 -15772.788,E2 -15772.788} C_VEL
LIN {X 0,Y 312.597,Z 334.169,A -85,B 0,C 180,E1 -15775.932,E2 -15775.932} C_VEL
LIN {X 0,Y 312.538,Z 334.178,A -85,B 0,C 180,E1 -15779.649,E2 -15779.649} C_VEL
LIN {X 0,Y 312.518,Z 334.18,A -85,B 0,C 180,E1 -15783.687,E2 -15783.687} C_VEL
LIN {X 0,Y 312.518,Z 334.182,A -85,B 0,C 180,E1 -15787.384,E2 -15787.384} C_VEL
LIN {X 0,Y 312.488,Z 334.184,A -85,B 0,C 180,E1 -15790.708,E2 -15790.708} C_VEL
LIN {X 0,Y 312.47,Z 334.184,A -85,B 0,C 180,E1 -15794.204,E2 -15794.204} C_VEL
LIN {X 0,Y 312.482,Z 334.183,A -85,B 0,C 180,E1 -15797.917,E2 -15797.917} C_VEL
LIN {X 0,Y 312.501,Z 334.18,A -85,B 0,C 180,E1 -15801.916,E2 -15801.916} C_VEL
LIN {X 0,Y 312.528,Z 334.178,A -85,B 0,C 180,E1 -15804.219,E2 -15804.219} C_VEL
LIN {X 0,Y 312.502,Z 334.182,A -85,B 0,C 180,E1 -15807.333,E2 -15807.333} C_VEL
LIN {X 0,Y 312.547,Z 334.176,A -85,B 0,C 180,E1 -15811.275,E2 -15811.275} C_VEL
LIN {X 0,Y 312.579,Z 334.176,A -85,B 0,C 180,E1 -15814.71,E2 -15814.71} C_VEL
LIN {X 0,Y 312.581,Z 334.171,A -85,B 0,C 180,E1 -15817.528,E2 -15817.528} C_VEL
LIN {X 0,Y 312.631,Z 334.164,A -85,B 0,C 180,E1 -15821.656,E2 -15821.656} C_VEL
LIN {X 0,Y 312.682,Z 334.157,A -85,B 0,C 180,E1 -15825.726,E2 -15825.726} C_VEL
LIN {X 0,Y 312.695,Z 334.156,A -85,B 0,C 180,E1 -15829.641,E2 -15829.641} C_VEL
LIN {X 0,Y 312.828,Z 334.14,A -85,B 0,C 180,E1 -15831.336,E2 -15831.336} C_VEL
LIN {X 0,Y 312.131,Z 334.231,A -85,B 0,C 180,E1 -15832.41,E2 -15832.41} C_VEL
LIN {X 0,Y 309.169,Z 334.598,A -85,B 0,C 180,E1 -15834.156,E2 -15834.156} C_VEL
LIN {X 0,Y 306.743,Z 334.898,A -85,B 0,C 180,E1 -15835.572,E2 -15835.572} C_VEL
LIN {X 0,Y 305.819,Z 335.016,A -85,B 0,C 180,E1 -15836.671,E2 -15836.671} C_VEL
LIN {X 0,Y 305.807,Z 335.013,A -85,B 0,C 180,E1 -15837.042,E2 -15837.042} C_VEL
LIN {X 0,Y 306.048,Z 334.986,A -85,B 0,C 180,E1 -15840,E2 -15840} C_VEL
LIN {X 0,Y 305.88,Z 335.008,A -85,B 0,C 180,E1 -15842.633,E2 -15842.633} C_VEL
LIN {X 0,Y 305.845,Z 335.012,A -85,B 0,C 180,E1 -15846.597,E2 -15846.597} C_VEL
LIN {X 0,Y 305.728,Z 335.024,A -85,B 0,C 180,E1 -15849.26,E2 -15849.26} C_VEL
LIN {X 0,Y 305.583,Z 335.042,A -85,B 0,C 180,E1 -15853.296,E2 -15853.296} C_VEL
LIN {X 0,Y 305.586,Z 335.046,A -85,B 0,C 180,E1 -15856.02,E2 -15856.02} C_VEL
LIN {X 0,Y 305.569,Z 335.044,A -85,B 0,C 180,E1 -15859.445,E2 -15859.445} C_VEL
LIN {X 0,Y 305.483,Z 335.055,A -85,B 0,C 180,E1 -15863.042,E2 -15863.042} C_VEL
LIN {X 0,Y 305.54,Z 335.05,A -85,B 0,C 180,E1 -15866.228,E2 -15866.228} C_VEL
LIN {X 0,Y 305.489,Z 335.054,A -85,B 0,C 180,E1 -15869.051,E2 -15869.051} C_VEL
LIN {X 0,Y 305.441,Z 335.065,A -85,B 0,C 180,E1 -15871.952,E2 -15871.952} C_VEL
LIN {X 0,Y 305.456,Z 335.059,A -85,B 0,C 180,E1 -15875.114,E2 -15875.114} C_VEL
LIN {X 0,Y 305.555,Z 335.231,A -85,B 0,C 180,E1 -15877.451,E2 -15877.451} C_VEL
LIN {X 0,Y 307.125,Z 343.611,A -85,B 0,C 180,E1 -15881.576,E2 -15881.576} C_VEL
LIN {X 0,Y 308.606,Z 351.14,A -85,B 0,C 180,E1 -15885.094,E2 -15885.094} C_VEL
LIN {X 0,Y 310.173,Z 358.472,A -85,B 0,C 180,E1 -15888.393,E2 -15888.393} C_VEL
LIN {X 0,Y 310.209,Z 361.68,A -85,B 0,C 180,E1 -15889.756,E2 -15889.756} C_VEL
LIN {X 0,Y 308.67,Z 371.331,A -85,B 0,C 180,E1 -15893.704,E2 -15893.704} C_VEL
LIN {X 0,Y 307.167,Z 382.633,A -85,B 0,C 180,E1 -15898.25,E2 -15898.25} C_VEL
LIN {X 0,Y 305.857,Z 395.186,A -85,B 0,C 180,E1 -15903.239,E2 -15903.239} C_VEL
LIN {X 0,Y 305.706,Z 397.247,A -85,B 0,C 180,E1 -15903.946,E2 -15903.946} C_VEL
LIN {X 0,Y 307.4,Z 416.858,A -85,B 0,C 180,E1 -15905.07,E2 -15905.07} C_VEL
LIN {X 0,Y 308.615,Z 431.511,A -85,B 0,C 180,E1 -15906.159,E2 -15906.159} C_VEL
LIN {X 0,Y 309.73,Z 445.376,A -85,B 0,C 180,E1 -15907.445,E2 -15907.445} C_VEL
LIN {X 0,Y 310.284,Z 455.712,A -85,B 0,C 180,E1 -15908.583,E2 -15908.583} C_VEL
LIN {X 0,Y 308.763,Z 468.47,A -85,B 0,C 180,E1 -15910.211,E2 -15910.211} C_VEL
LIN {X 0,Y 307.384,Z 480.013,A -85,B 0,C 180,E1 -15912.023,E2 -15912.023} C_VEL
LIN {X 0,Y 306.242,Z 490.472,A -85,B 0,C 180,E1 -15914.016,E2 -15914.016} C_VEL
LIN {X 0,Y 305.422,Z 499.17,A -85,B 0,C 180,E1 -15916.02,E2 -15916.02} C_VEL
LIN {X 0,Y 304.953,Z 507.536,A -85,B 0,C 180,E1 -15918.368,E2 -15918.368} C_VEL
LIN {X 0,Y 304.83,Z 514.199,A -85,B 0,C 180,E1 -15920.714,E2 -15920.714} C_VEL
LIN {X 0,Y 305.027,Z 518.632,A -85,B 0,C 180,E1 -15922.682,E2 -15922.682} C_VEL
LIN {X 0,Y 305.208,Z 522.188,A -85,B 0,C 180,E1 -15924.716,E2 -15924.716} C_VEL
LIN {X 0,Y 305.49,Z 525.347,A -85,B 0,C 180,E1 -15927.364,E2 -15927.364} C_VEL
LIN {X 0,Y 305.635,Z 526.324,A -85,B 0,C 180,E1 -15928.684,E2 -15928.684} C_VEL
LIN {X 0,Y 305.8,Z 526.911,A -85,B 0,C 180,E1 -15930.001,E2 -15930.001} C_VEL
LIN {X 0,Y 305.566,Z 527.042,A -85,B 0,C 180,E1 -15931.319,E2 -15931.319} C_VEL
LIN {X 0,Y 305.019,Z 526.162,A -85,B 0,C 180,E1 -15933.965,E2 -15933.965} C_VEL
LIN {X 0,Y 304.85,Z 525.178,A -85,B 0,C 180,E1 -15935.292,E2 -15935.292} C_VEL
LIN {X 0,Y 304.443,Z 522.095,A -85,B 0,C 180,E1 -15937.963,E2 -15937.963} C_VEL
LIN {X 0,Y 304.374,Z 517.574,A -85,B 0,C 180,E1 -15940.646,E2 -15940.646} C_VEL
LIN {X 0,Y 304.83,Z 511.579,A -85,B 0,C 180,E1 -15943.331,E2 -15943.331} C_VEL
LIN {X 0,Y 306.067,Z 504.054,A -85,B 0,C 180,E1 -15945.996,E2 -15945.996} C_VEL
LIN {X 0,Y 307.974,Z 494.873,A -85,B 0,C 180,E1 -15948.633,E2 -15948.633} C_VEL
LIN {X 0,Y 310.768,Z 483.845,A -85,B 0,C 180,E1 -15951.214,E2 -15951.214} C_VEL
LIN {X 0,Y 313.851,Z 472.723,A -85,B 0,C 180,E1 -15953.35,E2 -15953.35} C_VEL
LIN {X 0,Y 316.461,Z 462.967,A -85,B 0,C 180,E1 -15954.959,E2 -15954.959} C_VEL
LIN {X 0,Y 319.03,Z 449.216,A -85,B 0,C 180,E1 -15957.024,E2 -15957.024} C_VEL
LIN {X 0,Y 320.692,Z 437.381,A -85,B 0,C 180,E1 -15958.656,E2 -15958.656} C_VEL
LIN {X 0,Y 321.264,Z 424.826,A -85,B 0,C 180,E1 -15960.401,E2 -15960.401} C_VEL
LIN {X 0,Y 320.957,Z 413.31,A -85,B 0,C 180,E1 -15962.082,E2 -15962.082} C_VEL
LIN {X 0,Y 320.028,Z 402.553,A -85,B 0,C 180,E1 -15963.801,E2 -15963.801} C_VEL
LIN {X 0,Y 318.795,Z 392.904,A -85,B 0,C 180,E1 -15965.532,E2 -15965.532} C_VEL
LIN {X 0,Y 317.618,Z 384.629,A -85,B 0,C 180,E1 -15967.196,E2 -15967.196} C_VEL
LIN {X 0,Y 316.609,Z 377.991,A -85,B 0,C 180,E1 -15968.739,E2 -15968.739} C_VEL
LIN {X 0,Y 316.21,Z 374.911,A -85,B 0,C 180,E1 -15969.516,E2 -15969.516} C_VEL
LIN {X 0,Y 315.499,Z 368.209,A -85,B 0,C 180,E1 -15971.434,E2 -15971.434} C_VEL
LIN {X 0,Y 315.03,Z 365.482,A -85,B 0,C 180,E1 -15972.592,E2 -15972.592} C_VEL
LIN {X 0,Y 314.549,Z 362.579,A -85,B 0,C 180,E1 -15974.359,E2 -15974.359} C_VEL
LIN {X 0,Y 314.557,Z 360.55,A -85,B 0,C 180,E1 -15976.163,E2 -15976.163} C_VEL
LIN {X 0,Y 315.593,Z 359.375,A -85,B 0,C 180,E1 -15979.215,E2 -15979.215} C_VEL
LIN {X 0,Y 317.027,Z 359.113,A -85,B 0,C 180,E1 -15980.888,E2 -15980.888} C_VEL
LIN {X 0,Y 320.067,Z 360.746,A -85,B 0,C 180,E1 -15983.64,E2 -15983.64} C_VEL
LIN {X 0,Y 323.095,Z 363.274,A -85,B 0,C 180,E1 -15985.75,E2 -15985.75} C_VEL
LIN {X 0,Y 326.003,Z 366.686,A -85,B 0,C 180,E1 -15987.591,E2 -15987.591} C_VEL
LIN {X 0,Y 327.809,Z 371.054,A -85,B 0,C 180,E1 -15989.046,E2 -15989.046} C_VEL
LIN {X 0,Y 330.14,Z 379.033,A -85,B 0,C 180,E1 -15991.275,E2 -15991.275} C_VEL
LIN {X 0,Y 331.023,Z 384.102,A -85,B 0,C 180,E1 -15992.525,E2 -15992.525} C_VEL
LIN {X 0,Y 327.775,Z 395.248,A -85,B 0,C 180,E1 -15994.231,E2 -15994.231} C_VEL
LIN {X 0,Y 324.482,Z 405.244,A -85,B 0,C 180,E1 -15996.058,E2 -15996.058} C_VEL
LIN {X 0,Y 321.514,Z 413.418,A -85,B 0,C 180,E1 -15997.848,E2 -15997.848} C_VEL
LIN {X 0,Y 318.322,Z 421.493,A -85,B 0,C 180,E1 -15999.988,E2 -15999.988} C_VEL
LIN {X 0,Y 315.34,Z 428.8,A -85,B 0,C 180,E1 -16002.49,E2 -16002.49} C_VEL
LIN {X 0,Y 312.624,Z 434.793,A -85,B 0,C 180,E1 -16005.168,E2 -16005.168} C_VEL
LIN {X 0,Y 311.086,Z 437.822,A -85,B 0,C 180,E1 -16006.943,E2 -16006.943} C_VEL
LIN {X 0,Y 309.236,Z 440.999,A -85,B 0,C 180,E1 -16009.525,E2 -16009.525} C_VEL
LIN {X 0,Y 307.792,Z 442.844,A -85,B 0,C 180,E1 -16012.126,E2 -16012.126} C_VEL
LIN {X 0,Y 306.763,Z 443.391,A -85,B 0,C 180,E1 -16014.742,E2 -16014.742} C_VEL
LIN {X 0,Y 306.1,Z 442.628,A -85,B 0,C 180,E1 -16017.368,E2 -16017.368} C_VEL
LIN {X 0,Y 305.806,Z 440.534,A -85,B 0,C 180,E1 -16020,E2 -16020} C_VEL
LIN {X 0,Y 305.807,Z 438.97,A -85,B 0,C 180,E1 -16021.317,E2 -16021.317} C_VEL
LIN {X 0,Y 305.472,Z 434.83,A -85,B 0,C 180,E1 -16023.958,E2 -16023.958} C_VEL
LIN {X 0,Y 306.089,Z 429.13,A -85,B 0,C 180,E1 -16026.593,E2 -16026.593} C_VEL
LIN {X 0,Y 306.703,Z 421.803,A -85,B 0,C 180,E1 -16029.231,E2 -16029.231} C_VEL
LIN {X 0,Y 307.456,Z 413.79,A -85,B 0,C 180,E1 -16031.538,E2 -16031.538} C_VEL
LIN {X 0,Y 308.512,Z 403.988,A -85,B 0,C 180,E1 -16033.839,E2 -16033.839} C_VEL
LIN {X 0,Y 309.567,Z 393.894,A -85,B 0,C 180,E1 -16035.809,E2 -16035.809} C_VEL
LIN {X 0,Y 311.026,Z 381.796,A -85,B 0,C 180,E1 -16037.762,E2 -16037.762} C_VEL
LIN {X 0,Y 312.219,Z 369.689,A -85,B 0,C 180,E1 -16039.376,E2 -16039.376} C_VEL
LIN {X 0,Y 312.898,Z 362.462,A -85,B 0,C 180,E1 -16040.203,E2 -16040.203} C_VEL
LIN {X 0,Y 312.371,Z 359.319,A -85,B 0,C 180,E1 -16040.582,E2 -16040.582} C_VEL
LIN {X 0,Y 308.854,Z 346.961,A -85,B 0,C 180,E1 -16041.986,E2 -16041.986} C_VEL
LIN {X 0,Y 305.611,Z 335.616,A -85,B 0,C 180,E1 -16043.138,E2 -16043.138} C_VEL
LIN {X 0,Y 305.517,Z 335.102,A -85,B 0,C 180,E1 -16043.343,E2 -16043.343} C_VEL
LIN {X 0,Y 305.559,Z 335.048,A -85,B 0,C 180,E1 -16046.229,E2 -16046.229} C_VEL
LIN {X 0,Y 305.501,Z 335.055,A -85,B 0,C 180,E1 -16049.05,E2 -16049.05} C_VEL
LIN {X 0,Y 305.47,Z 335.056,A -85,B 0,C 180,E1 -16053.517,E2 -16053.517} C_VEL
LIN {X 0,Y 305.48,Z 335.058,A -85,B 0,C 180,E1 -16056.739,E2 -16056.739} C_VEL
LIN {X 0,Y 305.46,Z 335.062,A -85,B 0,C 180,E1 -16060.6,E2 -16060.6} C_VEL
LIN {X 0,Y 305.432,Z 335.061,A -85,B 0,C 180,E1 -16063.655,E2 -16063.655} C_VEL
LIN {X 0,Y 305.492,Z 335.053,A -85,B 0,C 180,E1 -16067.407,E2 -16067.407} C_VEL
LIN {X 0,Y 305.514,Z 335.051,A -85,B 0,C 180,E1 -16071.602,E2 -16071.602} C_VEL
LIN {X 0,Y 305.469,Z 335.057,A -85,B 0,C 180,E1 -16074.887,E2 -16074.887} C_VEL
LIN {X 0,Y 305.456,Z 335.062,A -85,B 0,C 180,E1 -16078.355,E2 -16078.355} C_VEL
LIN {X 0,Y 305.519,Z 335.05,A -85,B 0,C 180,E1 -16081.113,E2 -16081.113} C_VEL
LIN {X 0,Y 305.577,Z 335.048,A -85,B 0,C 180,E1 -16084.087,E2 -16084.087} C_VEL
LIN {X 0,Y 305.488,Z 335.056,A -85,B 0,C 180,E1 -16088.401,E2 -16088.401} C_VEL
LIN {X 0,Y 305.595,Z 335.04,A -85,B 0,C 180,E1 -16091.217,E2 -16091.217} C_VEL
LIN {X 0,Y 305.654,Z 335.034,A -85,B 0,C 180,E1 -16095.348,E2 -16095.348} C_VEL
LIN {X 0,Y 305.644,Z 335.036,A -85,B 0,C 180,E1 -16099.399,E2 -16099.399} C_VEL
LIN {X 0,Y 305.818,Z 335.017,A -85,B 0,C 180,E1 -16102.073,E2 -16102.073} C_VEL
LIN {X 0,Y 305.693,Z 335.029,A -85,B 0,C 180,E1 -16104.722,E2 -16104.722} C_VEL
LIN {X 0,Y 305.96,Z 334.995,A -85,B 0,C 180,E1 -16108.683,E2 -16108.683} C_VEL
LIN {X 0,Y 305.96,Z 334.997,A -85,B 0,C 180,E1 -16111.315,E2 -16111.315} C_VEL
LIN {X 0,Y 305.856,Z 335.008,A -85,B 0,C 180,E1 -16116.596,E2 -16116.596} C_VEL
LIN {X 0,Y 305.739,Z 335.025,A -85,B 0,C 180,E1 -16119.258,E2 -16119.258} C_VEL
LIN {X 0,Y 305.592,Z 335.044,A -85,B 0,C 180,E1 -16123.295,E2 -16123.295} C_VEL
LIN {X 0,Y 305.596,Z 335.042,A -85,B 0,C 180,E1 -16126.019,E2 -16126.019} C_VEL
LIN {X 0,Y 305.578,Z 335.048,A -85,B 0,C 180,E1 -16129.444,E2 -16129.444} C_VEL
LIN {X 0,Y 305.492,Z 335.056,A -85,B 0,C 180,E1 -16133.04,E2 -16133.04} C_VEL
LIN {X 0,Y 305.526,Z 335.049,A -85,B 0,C 180,E1 -16136.217,E2 -16136.217} C_VEL
LIN {X 0,Y 305.488,Z 335.057,A -85,B 0,C 180,E1 -16139.046,E2 -16139.046} C_VEL
LIN {X 0,Y 305.441,Z 335.06,A -85,B 0,C 180,E1 -16141.951,E2 -16141.951} C_VEL
LIN {X 0,Y 305.461,Z 335.062,A -85,B 0,C 180,E1 -16145.112,E2 -16145.112} C_VEL
LIN {X 0,Y 305.438,Z 335.061,A -85,B 0,C 180,E1 -16148.525,E2 -16148.525} C_VEL
LIN {X 0,Y 305.456,Z 335.059,A -85,B 0,C 180,E1 -16152.585,E2 -16152.585} C_VEL
LIN {X 0,Y 305.439,Z 335.061,A -85,B 0,C 180,E1 -16156.347,E2 -16156.347} C_VEL
LIN {X 0,Y 305.454,Z 335.058,A -85,B 0,C 180,E1 -16159.891,E2 -16159.891} C_VEL
LIN {X 0,Y 305.477,Z 335.056,A -85,B 0,C 180,E1 -16163.63,E2 -16163.63} C_VEL
LIN {X 0,Y 305.461,Z 335.059,A -85,B 0,C 180,E1 -16166.482,E2 -16166.482} C_VEL
LIN {X 0,Y 305.461,Z 335.058,A -85,B 0,C 180,E1 -16169.59,E2 -16169.59} C_VEL
LIN {X 0,Y 305.516,Z 335.054,A -85,B 0,C 180,E1 -16172.608,E2 -16172.608} C_VEL
LIN {X 0,Y 305.502,Z 335.052,A -85,B 0,C 180,E1 -16175.538,E2 -16175.538} C_VEL
LIN {X 0,Y 305.513,Z 335.051,A -85,B 0,C 180,E1 -16179.814,E2 -16179.814} C_VEL
LIN {X 0,Y 305.568,Z 335.049,A -85,B 0,C 180,E1 -16182.602,E2 -16182.602} C_VEL
LIN {X 0,Y 305.642,Z 335.035,A -85,B 0,C 180,E1 -16185.348,E2 -16185.348} C_VEL
LIN {X 0,Y 305.631,Z 335.036,A -85,B 0,C 180,E1 -16189.399,E2 -16189.399} C_VEL
LIN {X 0,Y 305.807,Z 335.016,A -85,B 0,C 180,E1 -16192.074,E2 -16192.074} C_VEL
LIN {X 0,Y 305.683,Z 335.033,A -85,B 0,C 180,E1 -16194.723,E2 -16194.723} C_VEL
LIN {X 0,Y 305.807,Z 335.013,A -85,B 0,C 180,E1 -16197.042,E2 -16197.042} C_VEL
LIN {X 0,Y 305.337,Z 335.076,A -85,B 0,C 180,E1 -16198.142,E2 -16198.142} C_VEL
LIN {X 0,Y 303.875,Z 335.261,A -85,B 0,C 180,E1 -16199.223,E2 -16199.223} C_VEL
LIN {X 0,Y 299.237,Z 335.837,A -85,B 0,C 180,E1 -16202.135,E2 -16202.135} C_VEL
LIN {X 0,Y 298.785,Z 335.89,A -85,B 0,C 180,E1 -16202.896,E2 -16202.896} C_VEL
LIN {X 0,Y 298.79,Z 335.89,A -85,B 0,C 180,E1 -16206.754,E2 -16206.754} C_VEL
LIN {X 0,Y 298.673,Z 335.903,A -85,B 0,C 180,E1 -16209.48,E2 -16209.48} C_VEL
LIN {X 0,Y 298.546,Z 335.92,A -85,B 0,C 180,E1 -16213.615,E2 -16213.615} C_VEL
LIN {X 0,Y 298.541,Z 335.922,A -85,B 0,C 180,E1 -16216.409,E2 -16216.409} C_VEL
LIN {X 0,Y 298.504,Z 335.925,A -85,B 0,C 180,E1 -16219.655,E2 -16219.655} C_VEL
LIN {X 0,Y 298.45,Z 335.933,A -85,B 0,C 180,E1 -16223.598,E2 -16223.598} C_VEL
LIN {X 0,Y 298.482,Z 335.927,A -85,B 0,C 180,E1 -16226.575,E2 -16226.575} C_VEL
LIN {X 0,Y 298.415,Z 335.938,A -85,B 0,C 180,E1 -16229.641,E2 -16229.641} C_VEL
LIN {X 0,Y 298.391,Z 335.939,A -85,B 0,C 180,E1 -16232.8,E2 -16232.8} C_VEL
LIN {X 0,Y 298.478,Z 336.013,A -85,B 0,C 180,E1 -16237.056,E2 -16237.056} C_VEL
LIN {X 0,Y 299.956,Z 343.782,A -85,B 0,C 180,E1 -16240.998,E2 -16240.998} C_VEL
LIN {X 0,Y 301.599,Z 352.232,A -85,B 0,C 180,E1 -16245.052,E2 -16245.052} C_VEL
LIN {X 0,Y 303.241,Z 360.347,A -85,B 0,C 180,E1 -16248.768,E2 -16248.768} C_VEL
LIN {X 0,Y 302.852,Z 364.509,A -85,B 0,C 180,E1 -16250.55,E2 -16250.55} C_VEL
LIN {X 0,Y 301.173,Z 374.606,A -85,B 0,C 180,E1 -16254.759,E2 -16254.759} C_VEL
LIN {X 0,Y 299.864,Z 384.809,A -85,B 0,C 180,E1 -16258.963,E2 -16258.963} C_VEL
LIN {X 0,Y 298.678,Z 396.184,A -85,B 0,C 180,E1 -16263.539,E2 -16263.539} C_VEL
LIN {X 0,Y 298.985,Z 400.588,A -85,B 0,C 180,E1 -16263.827,E2 -16263.827} C_VEL
LIN {X 0,Y 300.299,Z 415.773,A -85,B 0,C 180,E1 -16264.717,E2 -16264.717} C_VEL
LIN {X 0,Y 301.565,Z 431.65,A -85,B 0,C 180,E1 -16265.936,E2 -16265.936} C_VEL
LIN {X 0,Y 302.665,Z 445.495,A -85,B 0,C 180,E1 -16267.28,E2 -16267.28} C_VEL
LIN {X 0,Y 303.226,Z 455.44,A -85,B 0,C 180,E1 -16268.413,E2 -16268.413} C_VEL
LIN {X 0,Y 301.713,Z 468.031,A -85,B 0,C 180,E1 -16270.084,E2 -16270.084} C_VEL
LIN {X 0,Y 300.322,Z 479.453,A -85,B 0,C 180,E1 -16271.938,E2 -16271.938} C_VEL
LIN {X 0,Y 299.181,Z 489.886,A -85,B 0,C 180,E1 -16273.994,E2 -16273.994} C_VEL
LIN {X 0,Y 298.36,Z 498.432,A -85,B 0,C 180,E1 -16276.03,E2 -16276.03} C_VEL
LIN {X 0,Y 297.916,Z 506.727,A -85,B 0,C 180,E1 -16278.434,E2 -16278.434} C_VEL
LIN {X 0,Y 297.819,Z 512.456,A -85,B 0,C 180,E1 -16280.493,E2 -16280.493} C_VEL
LIN {X 0,Y 298.018,Z 517.143,A -85,B 0,C 180,E1 -16282.568,E2 -16282.568} C_VEL
LIN {X 0,Y 298.199,Z 520.705,A -85,B 0,C 180,E1 -16284.592,E2 -16284.592} C_VEL
LIN {X 0,Y 298.502,Z 523.981,A -85,B 0,C 180,E1 -16287.302,E2 -16287.302} C_VEL
LIN {X 0,Y 298.661,Z 525.012,A -85,B 0,C 180,E1 -16288.653,E2 -16288.653} C_VEL
LIN {X 0,Y 298.828,Z 525.653,A -85,B 0,C 180,E1 -16290.001,E2 -16290.001} C_VEL
LIN {X 0,Y 298.545,Z 525.828,A -85,B 0,C 180,E1 -16291.35,E2 -16291.35} C_VEL
LIN {X 0,Y 297.969,Z 525.049,A -85,B 0,C 180,E1 -16294.059,E2 -16294.059} C_VEL
LIN {X 0,Y 297.788,Z 524.121,A -85,B 0,C 180,E1 -16295.418,E2 -16295.418} C_VEL
LIN {X 0,Y 297.365,Z 521.152,A -85,B 0,C 180,E1 -16298.154,E2 -16298.154} C_VEL
LIN {X 0,Y 297.299,Z 516.77,A -85,B 0,C 180,E1 -16300.902,E2 -16300.902} C_VEL
LIN {X 0,Y 297.826,Z 510.966,A -85,B 0,C 180,E1 -16303.65,E2 -16303.65} C_VEL
LIN {X 0,Y 299.154,Z 503.683,A -85,B 0,C 180,E1 -16306.376,E2 -16306.376} C_VEL
LIN {X 0,Y 301.189,Z 494.756,A -85,B 0,C 180,E1 -16309.068,E2 -16309.068} C_VEL
LIN {X 0,Y 304.142,Z 484.034,A -85,B 0,C 180,E1 -16311.7,E2 -16311.7} C_VEL
LIN {X 0,Y 307.003,Z 474.383,A -85,B 0,C 180,E1 -16313.674,E2 -16313.674} C_VEL
LIN {X 0,Y 310.087,Z 463.927,A -85,B 0,C 180,E1 -16315.509,E2 -16315.509} C_VEL
LIN {X 0,Y 313.117,Z 449.724,A -85,B 0,C 180,E1 -16317.759,E2 -16317.759} C_VEL
LIN {X 0,Y 314.905,Z 438.439,A -85,B 0,C 180,E1 -16319.407,E2 -16319.407} C_VEL
LIN {X 0,Y 315.713,Z 427.753,A -85,B 0,C 180,E1 -16320.994,E2 -16320.994} C_VEL
LIN {X 0,Y 315.778,Z 417.085,A -85,B 0,C 180,E1 -16322.65,E2 -16322.65} C_VEL
LIN {X 0,Y 315.309,Z 406.455,A -85,B 0,C 180,E1 -16324.442,E2 -16324.442} C_VEL
LIN {X 0,Y 314.389,Z 396.145,A -85,B 0,C 180,E1 -16326.413,E2 -16326.413} C_VEL
LIN {X 0,Y 313.647,Z 388.919,A -85,B 0,C 180,E1 -16327.975,E2 -16327.975} C_VEL
LIN {X 0,Y 312.989,Z 381.018,A -85,B 0,C 180,E1 -16329.885,E2 -16329.885} C_VEL
LIN {X 0,Y 312.556,Z 373.63,A -85,B 0,C 180,E1 -16332.096,E2 -16332.096} C_VEL
LIN {X 0,Y 312.057,Z 370.163,A -85,B 0,C 180,E1 -16333.889,E2 -16333.889} C_VEL
LIN {X 0,Y 312.012,Z 367.33,A -85,B 0,C 180,E1 -16336.121,E2 -16336.121} C_VEL
LIN {X 0,Y 312.334,Z 366.423,A -85,B 0,C 180,E1 -16337.95,E2 -16337.95} C_VEL
LIN {X 0,Y 313.29,Z 365.824,A -85,B 0,C 180,E1 -16339.706,E2 -16339.706} C_VEL
LIN {X 0,Y 314.708,Z 365.905,A -85,B 0,C 180,E1 -16341.41,E2 -16341.41} C_VEL
LIN {X 0,Y 316.46,Z 366.857,A -85,B 0,C 180,E1 -16343.157,E2 -16343.157} C_VEL
LIN {X 0,Y 318.816,Z 368.65,A -85,B 0,C 180,E1 -16345.03,E2 -16345.03} C_VEL
LIN {X 0,Y 321.342,Z 371.47,A -85,B 0,C 180,E1 -16346.855,E2 -16346.855} C_VEL
LIN {X 0,Y 322.458,Z 373.355,A -85,B 0,C 180,E1 -16347.707,E2 -16347.707} C_VEL
LIN {X 0,Y 324.216,Z 379.143,A -85,B 0,C 180,E1 -16349.599,E2 -16349.599} C_VEL
LIN {X 0,Y 325.482,Z 385.4,A -85,B 0,C 180,E1 -16351.358,E2 -16351.358} C_VEL
LIN {X 0,Y 325.672,Z 388.004,A -85,B 0,C 180,E1 -16352.007,E2 -16352.007} C_VEL
LIN {X 0,Y 322.03,Z 398.915,A -85,B 0,C 180,E1 -16353.737,E2 -16353.737} C_VEL
LIN {X 0,Y 318.609,Z 408.382,A -85,B 0,C 180,E1 -16355.569,E2 -16355.569} C_VEL
LIN {X 0,Y 314.965,Z 417.439,A -85,B 0,C 180,E1 -16357.708,E2 -16357.708} C_VEL
LIN {X 0,Y 312.072,Z 423.995,A -85,B 0,C 180,E1 -16359.57,E2 -16359.57} C_VEL
LIN {X 0,Y 308.907,Z 431.016,A -85,B 0,C 180,E1 -16362.113,E2 -16362.113} C_VEL
LIN {X 0,Y 306.412,Z 436.01,A -85,B 0,C 180,E1 -16364.439,E2 -16364.439} C_VEL
LIN {X 0,Y 304.405,Z 439.616,A -85,B 0,C 180,E1 -16366.652,E2 -16366.652} C_VEL
LIN {X 0,Y 302.454,Z 442.6,A -85,B 0,C 180,E1 -16369.287,E2 -16369.287} C_VEL
LIN {X 0,Y 300.903,Z 444.274,A -85,B 0,C 180,E1 -16371.944,E2 -16371.944} C_VEL
LIN {X 0,Y 299.803,Z 444.654,A -85,B 0,C 180,E1 -16374.62,E2 -16374.62} C_VEL
LIN {X 0,Y 299.089,Z 443.715,A -85,B 0,C 180,E1 -16377.307,E2 -16377.307} C_VEL
LIN {X 0,Y 298.783,Z 441.43,A -85,B 0,C 180,E1 -16380,E2 -16380} C_VEL
LIN {X 0,Y 298.782,Z 439.782,A -85,B 0,C 180,E1 -16381.348,E2 -16381.348} C_VEL
LIN {X 0,Y 298.431,Z 435.489,A -85,B 0,C 180,E1 -16384.052,E2 -16384.052} C_VEL
LIN {X 0,Y 299.061,Z 429.633,A -85,B 0,C 180,E1 -16386.748,E2 -16386.748} C_VEL
LIN {X 0,Y 299.605,Z 423.14,A -85,B 0,C 180,E1 -16389.111,E2 -16389.111} C_VEL
LIN {X 0,Y 300.363,Z 415.192,A -85,B 0,C 180,E1 -16391.472,E2 -16391.472} C_VEL
LIN {X 0,Y 301.446,Z 405.456,A -85,B 0,C 180,E1 -16393.826,E2 -16393.826} C_VEL
LIN {X 0,Y 302.492,Z 395.418,A -85,B 0,C 180,E1 -16395.843,E2 -16395.843} C_VEL
LIN {X 0,Y 303.926,Z 383.414,A -85,B 0,C 180,E1 -16397.842,E2 -16397.842} C_VEL
LIN {X 0,Y 305.198,Z 371.381,A -85,B 0,C 180,E1 -16399.506,E2 -16399.506} C_VEL
LIN {X 0,Y 305.976,Z 363.178,A -85,B 0,C 180,E1 -16400.469,E2 -16400.469} C_VEL
LIN {X 0,Y 302.891,Z 351.639,A -85,B 0,C 180,E1 -16401.854,E2 -16401.854} C_VEL
LIN {X 0,Y 298.649,Z 336.855,A -85,B 0,C 180,E1 -16403.395,E2 -16403.395} C_VEL
LIN {X 0,Y 298.506,Z 335.966,A -85,B 0,C 180,E1 -16403.686,E2 -16403.686} C_VEL
LIN {X 0,Y 298.497,Z 335.93,A -85,B 0,C 180,E1 -16406.574,E2 -16406.574} C_VEL
LIN {X 0,Y 298.426,Z 335.934,A -85,B 0,C 180,E1 -16409.641,E2 -16409.641} C_VEL
LIN {X 0,Y 298.401,Z 335.941,A -85,B 0,C 180,E1 -16412.8,E2 -16412.8} C_VEL
LIN {X 0,Y 298.452,Z 335.933,A -85,B 0,C 180,E1 -16416.807,E2 -16416.807} C_VEL
LIN {X 0,Y 298.392,Z 335.939,A -85,B 0,C 180,E1 -16421.087,E2 -16421.087} C_VEL
LIN {X 0,Y 298.404,Z 335.937,A -85,B 0,C 180,E1 -16423.103,E2 -16423.103} C_VEL
LIN {X 0,Y 298.438,Z 335.933,A -85,B 0,C 180,E1 -16426.926,E2 -16426.926} C_VEL
LIN {X 0,Y 298.431,Z 335.934,A -85,B 0,C 180,E1 -16431.001,E2 -16431.001} C_VEL
LIN {X 0,Y 298.44,Z 335.934,A -85,B 0,C 180,E1 -16433.932,E2 -16433.932} C_VEL
LIN {X 0,Y 298.4,Z 335.94,A -85,B 0,C 180,E1 -16437.983,E2 -16437.983} C_VEL
LIN {X 0,Y 298.464,Z 335.932,A -85,B 0,C 180,E1 -16441.903,E2 -16441.903} C_VEL
LIN {X 0,Y 298.489,Z 335.926,A -85,B 0,C 180,E1 -16444.923,E2 -16444.923} C_VEL
LIN {X 0,Y 298.446,Z 335.931,A -85,B 0,C 180,E1 -16449.314,E2 -16449.314} C_VEL
LIN {X 0,Y 298.543,Z 335.923,A -85,B 0,C 180,E1 -16452.179,E2 -16452.179} C_VEL
LIN {X 0,Y 298.599,Z 335.912,A -85,B 0,C 180,E1 -16454.994,E2 -16454.994} C_VEL
LIN {X 0,Y 298.599,Z 335.912,A -85,B 0,C 180,E1 -16459.146,E2 -16459.146} C_VEL
LIN {X 0,Y 298.764,Z 335.897,A -85,B 0,C 180,E1 -16461.885,E2 -16461.885} C_VEL
LIN {X 0,Y 298.665,Z 335.904,A -85,B 0,C 180,E1 -16464.598,E2 -16464.598} C_VEL
LIN {X 0,Y 298.927,Z 335.871,A -85,B 0,C 180,E1 -16468.652,E2 -16468.652} C_VEL
LIN {X 0,Y 298.927,Z 335.874,A -85,B 0,C 180,E1 -16471.346,E2 -16471.346} C_VEL
LIN {X 0,Y 298.802,Z 335.886,A -85,B 0,C 180,E1 -16476.753,E2 -16476.753} C_VEL
LIN {X 0,Y 298.684,Z 335.906,A -85,B 0,C 180,E1 -16479.479,E2 -16479.479} C_VEL
LIN {X 0,Y 298.555,Z 335.922,A -85,B 0,C 180,E1 -16483.614,E2 -16483.614} C_VEL
LIN {X 0,Y 298.551,Z 335.918,A -85,B 0,C 180,E1 -16486.407,E2 -16486.407} C_VEL
LIN {X 0,Y 298.513,Z 335.926,A -85,B 0,C 180,E1 -16489.653,E2 -16489.653} C_VEL
LIN {X 0,Y 298.458,Z 335.933,A -85,B 0,C 180,E1 -16493.596,E2 -16493.596} C_VEL
LIN {X 0,Y 298.485,Z 335.927,A -85,B 0,C 180,E1 -16496.573,E2 -16496.573} C_VEL
LIN {X 0,Y 298.416,Z 335.937,A -85,B 0,C 180,E1 -16499.64,E2 -16499.64} C_VEL
LIN {X 0,Y 298.394,Z 335.939,A -85,B 0,C 180,E1 -16502.799,E2 -16502.799} C_VEL
LIN {X 0,Y 298.442,Z 335.934,A -85,B 0,C 180,E1 -16506.806,E2 -16506.806} C_VEL
LIN {X 0,Y 298.386,Z 335.943,A -85,B 0,C 180,E1 -16511.086,E2 -16511.086} C_VEL
LIN {X 0,Y 298.385,Z 335.944,A -85,B 0,C 180,E1 -16515.04,E2 -16515.04} C_VEL
